// TIA Portal V18 export
FUNCTION "ST10_Output" : Void   // FC1002, LAD
{ S7_Optimized_Access := 'FALSE' }
VERSION : 0.1
// stored: AutoNumber false, IsIECCheckEnabled false, SetENOAutomatically false, UDAEnableTagReadback false
   VAR_TEMP   // added for the SCL form of the ladder/FBD networks
      _w1 : Bool;
      _w2 : Bool;
      _w3 : Bool;
      _w4 : Bool;
      _w5 : Bool;
      _w6 : Bool;
   END_VAR
BEGIN

REGION Network 1 (SCL): 安全门锁定信号映射SafetyDoorCoil
   "oSafetyDoorLocked_1" := "ST10_SysOutput".SafetyDoorCoil[1];
   "oSafetyDoorLocked_2" := "ST10_SysOutput".SafetyDoorCoil[2];
   "oSafetyDoorLocked_3" := "ST10_SysOutput".SafetyDoorCoil[3];
   "oSafetyDoorLocked_4" := "ST10_SysOutput".SafetyDoorCoil[4];
   "oSafetyDoorLocked_5" := "ST10_SysOutput".SafetyDoorCoil[5];
   "oSafetyDoorLocked_6" := "ST10_SysOutput".SafetyDoorCoil[6];
   "oSafetyDoorLocked_7" := "ST10_SysOutput".SafetyDoorCoil[7];
   "oSafetyDoorLocked_8" := "ST10_SysOutput".SafetyDoorCoil[8];
   "oSafetyDoorLocked" := "ST10_SysOutput".SafetyDoorCoil[9];
END_REGION

REGION Network 2 (SCL): 安全门锁定信号映射SafetyDoorCoil
   "oMaterielDoorLocked_H1" := "ST10_SysOutput".MaterialDoorCoil[1];
   "oMaterielDoorLocked_H2" := "ST10_SysOutput".MaterialDoorCoil[2];
   "oMaterielDoorLocked_J1" := "ST10_SysOutput".MaterialDoorCoil[3];
   "oMaterielDoorLocked_J2" := "ST10_SysOutput".MaterialDoorCoil[4];
   "oMaterielDoorLocked_K1" := "ST10_SysOutput".MaterialDoorCoil[5];
   "oMaterielDoorLocked_K2" := "ST10_SysOutput".MaterialDoorCoil[6];
   "oMaterielDoorLocked_L1" := "ST10_SysOutput".MaterialDoorCoil[7];


   "oE-NG-01SafetyGate" := "ST10_SysOutput".MaterialDoorCoil[8];
   "oE-NG-02SafetyGate" := "ST10_SysOutput".MaterialDoorCoil[9];
END_REGION

REGION Network 3: 塔灯
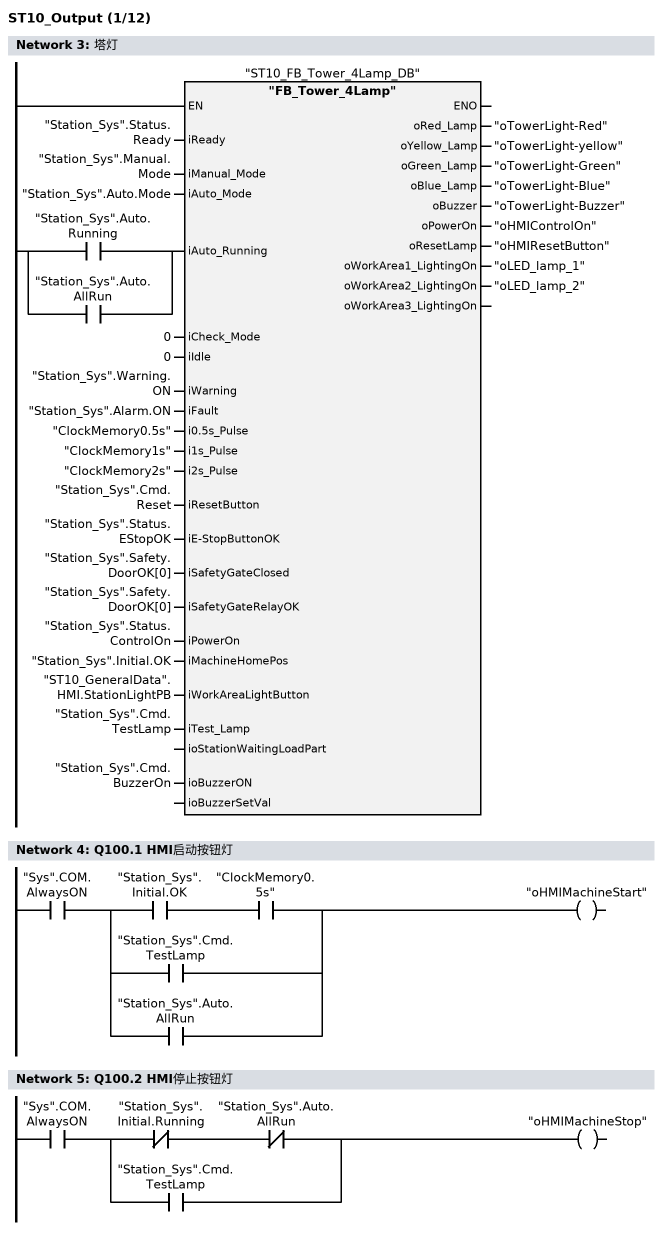
   RUNG wire#powerrail
      "ST10_FB_Tower_4Lamp_DB"(iAuto_Running := wire#w1, iReady := "Station_Sys".Status.Ready, iManual_Mode := "Station_Sys".Manual.Mode, iAuto_Mode := "Station_Sys".Auto.Mode, iCheck_Mode := 0, iIdle := 0, iWarning := "Station_Sys".Warning.ON, iFault := "Station_Sys".Alarm.ON, "i0.5s_Pulse" := "ClockMemory0.5s", i1s_Pulse := "ClockMemory1s", i2s_Pulse := "ClockMemory2s", iResetButton := "Station_Sys".Cmd.Reset, "iE-StopButtonOK" := "Station_Sys".Status.EStopOK, iSafetyGateClosed := "Station_Sys".Safety.DoorOK[0], iSafetyGateRelayOK := "Station_Sys".Safety.DoorOK[0], iPowerOn := "Station_Sys".Status.ControlOn, iMachineHomePos := "Station_Sys".Initial.OK, iWorkAreaLightButton := "ST10_GeneralData".HMI.StationLightPB, iTest_Lamp := "Station_Sys".Cmd.TestLamp, ioStationWaitingLoadPart :=, ioBuzzerON := "Station_Sys".Cmd.BuzzerOn, ioBuzzerSetVal :=, oRed_Lamp => "oTowerLight-Red", oYellow_Lamp => "oTowerLight-yellow", oGreen_Lamp => "oTowerLight-Green", oBlue_Lamp => "oTowerLight-Blue", oBuzzer => "oTowerLight-Buzzer", oPowerOn => "oHMIControlOn", oResetLamp => "oHMIResetButton", oWorkArea1_LightingOn => "oLED_lamp_1", oWorkArea2_LightingOn => "oLED_lamp_2", oWorkArea3_LightingOn =>)
   END_RUNG
   RUNG wire#powerrail
      Contact( "Station_Sys".Auto.Running )
   END_RUNG wire#w1
   RUNG wire#powerrail
      Contact( "Station_Sys".Auto.AllRun )
   END_RUNG wire#w1
   // the same network as SCL:
   "ST10_FB_Tower_4Lamp_DB"(iReady := "Station_Sys".Status.Ready,   // "FB_Tower_4Lamp"
                           iManual_Mode := "Station_Sys".Manual.Mode,
                           iAuto_Mode := "Station_Sys".Auto.Mode,
                           iAuto_Running := "Station_Sys".Auto.Running OR "Station_Sys".Auto.AllRun,
                           iCheck_Mode := 0,
                           iIdle := 0,
                           iWarning := "Station_Sys".Warning.ON,
                           iFault := "Station_Sys".Alarm.ON,
                           "i0.5s_Pulse" := "ClockMemory0.5s",
                           i1s_Pulse := "ClockMemory1s",
                           i2s_Pulse := "ClockMemory2s",
                           iResetButton := "Station_Sys".Cmd.Reset,
                           "iE-StopButtonOK" := "Station_Sys".Status.EStopOK,
                           iSafetyGateClosed := "Station_Sys".Safety.DoorOK[0],
                           iSafetyGateRelayOK := "Station_Sys".Safety.DoorOK[0],
                           iPowerOn := "Station_Sys".Status.ControlOn,
                           iMachineHomePos := "Station_Sys".Initial.OK,
                           iWorkAreaLightButton := "ST10_GeneralData".HMI.StationLightPB,
                           iTest_Lamp := "Station_Sys".Cmd.TestLamp,
                           ioBuzzerON := "Station_Sys".Cmd.BuzzerOn,
                           oRed_Lamp => "oTowerLight-Red",
                           oYellow_Lamp => "oTowerLight-yellow",
                           oGreen_Lamp => "oTowerLight-Green",
                           oBlue_Lamp => "oTowerLight-Blue",
                           oBuzzer => "oTowerLight-Buzzer",
                           oPowerOn => "oHMIControlOn",
                           oResetLamp => "oHMIResetButton",
                           oWorkArea1_LightingOn => "oLED_lamp_1",
                           oWorkArea2_LightingOn => "oLED_lamp_2");
END_REGION

REGION Network 4: Q100.1 HMI启动按钮灯
   RUNG wire#powerrail
      Contact( "Sys".COM.AlwaysON )
      wire#w1
      Contact( "Station_Sys".Initial.OK )
      Contact( "ClockMemory0.5s" )
      wire#w2
      Coil( "oHMIMachineStart" )
   END_RUNG
   RUNG wire#w1
      Contact( "Station_Sys".Cmd.TestLamp )
   END_RUNG wire#w2
   RUNG wire#w1
      Contact( "Station_Sys".Auto.AllRun )
   END_RUNG wire#w2
   // the same network as SCL:
   "oHMIMachineStart" := "Sys".COM.AlwaysON AND (("Station_Sys".Initial.OK AND "ClockMemory0.5s") OR "Station_Sys".Cmd.TestLamp OR "Station_Sys".Auto.AllRun);
END_REGION

REGION Network 5: Q100.2 HMI停止按钮灯
   RUNG wire#powerrail
      Contact( "Sys".COM.AlwaysON )
      wire#w1
      I_Contact( "Station_Sys".Initial.Running )
      I_Contact( "Station_Sys".Auto.AllRun )
      wire#w2
      Coil( "oHMIMachineStop" )
   END_RUNG
   RUNG wire#w1
      Contact( "Station_Sys".Cmd.TestLamp )
   END_RUNG wire#w2
   // the same network as SCL:
   "oHMIMachineStop" := "Sys".COM.AlwaysON AND ((NOT "Station_Sys".Initial.Running AND NOT "Station_Sys".Auto.AllRun) OR "Station_Sys".Cmd.TestLamp);
END_REGION

REGION Network 6: Q100.4 HMI开门按钮灯
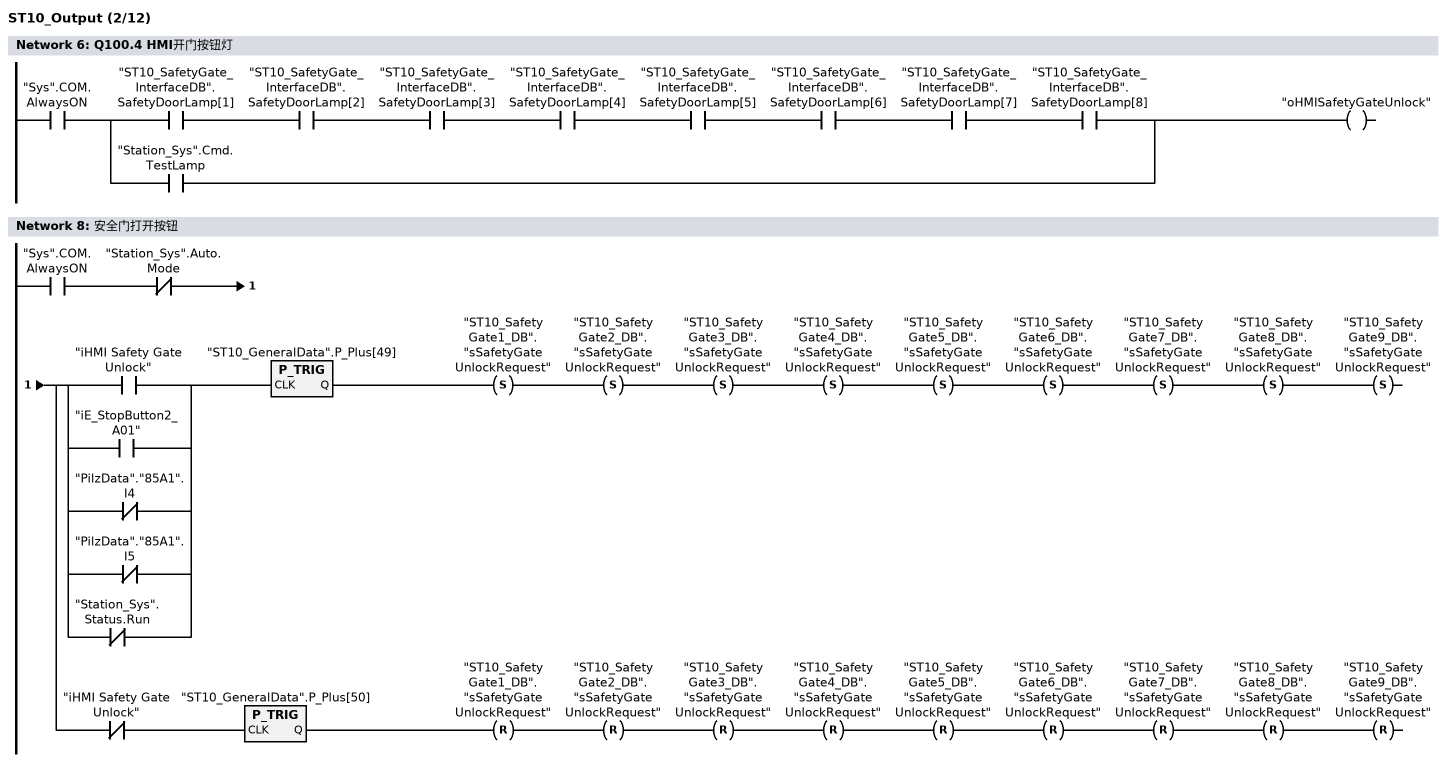
   RUNG wire#powerrail
      Contact( "Sys".COM.AlwaysON )
      wire#w1
      Contact( "ST10_SafetyGate_InterfaceDB".SafetyDoorLamp[1] )
      Contact( "ST10_SafetyGate_InterfaceDB".SafetyDoorLamp[2] )
      Contact( "ST10_SafetyGate_InterfaceDB".SafetyDoorLamp[3] )
      Contact( "ST10_SafetyGate_InterfaceDB".SafetyDoorLamp[4] )
      Contact( "ST10_SafetyGate_InterfaceDB".SafetyDoorLamp[5] )
      Contact( "ST10_SafetyGate_InterfaceDB".SafetyDoorLamp[6] )
      Contact( "ST10_SafetyGate_InterfaceDB".SafetyDoorLamp[7] )
      Contact( "ST10_SafetyGate_InterfaceDB".SafetyDoorLamp[8] )
      wire#w2
      Coil( "oHMISafetyGateUnlock" )
   END_RUNG
   RUNG wire#w1
      Contact( "Station_Sys".Cmd.TestLamp )
   END_RUNG wire#w2
   // the same network as SCL:
   "oHMISafetyGateUnlock" := "Sys".COM.AlwaysON AND (("ST10_SafetyGate_InterfaceDB".SafetyDoorLamp[1] AND "ST10_SafetyGate_InterfaceDB".SafetyDoorLamp[2] AND "ST10_SafetyGate_InterfaceDB".SafetyDoorLamp[3] AND "ST10_SafetyGate_InterfaceDB".SafetyDoorLamp[4] AND "ST10_SafetyGate_InterfaceDB".SafetyDoorLamp[5] AND "ST10_SafetyGate_InterfaceDB".SafetyDoorLamp[6] AND "ST10_SafetyGate_InterfaceDB".SafetyDoorLamp[7] AND "ST10_SafetyGate_InterfaceDB".SafetyDoorLamp[8]) OR "Station_Sys".Cmd.TestLamp);
END_REGION

REGION Network 8: 安全门打开按钮
   RUNG wire#powerrail
      Contact( "Sys".COM.AlwaysON )
      I_Contact( "Station_Sys".Auto.Mode )
      wire#w1
      Contact( "iHMI Safety Gate Unlock" )
      wire#w2
      P_Trig( "ST10_GeneralData".P_Plus[49] )
      S_Coil( "ST10_SafetyGate1_DB"."sSafetyGate UnlockRequest" )
      S_Coil( "ST10_SafetyGate2_DB"."sSafetyGate UnlockRequest" )
      S_Coil( "ST10_SafetyGate3_DB"."sSafetyGate UnlockRequest" )
      S_Coil( "ST10_SafetyGate4_DB"."sSafetyGate UnlockRequest" )
      S_Coil( "ST10_SafetyGate5_DB"."sSafetyGate UnlockRequest" )
      S_Coil( "ST10_SafetyGate6_DB"."sSafetyGate UnlockRequest" )
      S_Coil( "ST10_SafetyGate7_DB"."sSafetyGate UnlockRequest" )
      S_Coil( "ST10_SafetyGate8_DB"."sSafetyGate UnlockRequest" )
      S_Coil( "ST10_SafetyGate9_DB"."sSafetyGate UnlockRequest" )
   END_RUNG
   RUNG wire#w1
      Contact( "iE_StopButton2_A01" )
   END_RUNG wire#w2
   RUNG wire#w1
      I_Contact( "PilzData"."85A1".I4 )
   END_RUNG wire#w2
   RUNG wire#w1
      I_Contact( "PilzData"."85A1".I5 )
   END_RUNG wire#w2
   RUNG wire#w1
      I_Contact( "Station_Sys".Status.Run )
   END_RUNG wire#w2
   RUNG wire#w1
      I_Contact( "iHMI Safety Gate Unlock" )
      P_Trig( "ST10_GeneralData".P_Plus[50] )
      R_Coil( "ST10_SafetyGate1_DB"."sSafetyGate UnlockRequest" )
      R_Coil( "ST10_SafetyGate2_DB"."sSafetyGate UnlockRequest" )
      R_Coil( "ST10_SafetyGate3_DB"."sSafetyGate UnlockRequest" )
      R_Coil( "ST10_SafetyGate4_DB"."sSafetyGate UnlockRequest" )
      R_Coil( "ST10_SafetyGate5_DB"."sSafetyGate UnlockRequest" )
      R_Coil( "ST10_SafetyGate6_DB"."sSafetyGate UnlockRequest" )
      R_Coil( "ST10_SafetyGate7_DB"."sSafetyGate UnlockRequest" )
      R_Coil( "ST10_SafetyGate8_DB"."sSafetyGate UnlockRequest" )
      R_Coil( "ST10_SafetyGate9_DB"."sSafetyGate UnlockRequest" )
   END_RUNG
   // the same network as SCL:
   #_w1 := "Sys".COM.AlwaysON AND NOT "Station_Sys".Auto.Mode;
   #_w2 := #_w1 AND ("iHMI Safety Gate Unlock" OR "iE_StopButton2_A01" OR NOT "PilzData"."85A1".I4 OR NOT "PilzData"."85A1".I5 OR NOT "Station_Sys".Status.Run);
   #_w3 := #_w2 AND NOT "ST10_GeneralData".P_Plus[49];   // rising edge
   "ST10_GeneralData".P_Plus[49] := #_w2;
   IF #_w3 THEN
       "ST10_SafetyGate1_DB"."sSafetyGate UnlockRequest" := TRUE;
       "ST10_SafetyGate2_DB"."sSafetyGate UnlockRequest" := TRUE;
       "ST10_SafetyGate3_DB"."sSafetyGate UnlockRequest" := TRUE;
       "ST10_SafetyGate4_DB"."sSafetyGate UnlockRequest" := TRUE;
       "ST10_SafetyGate5_DB"."sSafetyGate UnlockRequest" := TRUE;
       "ST10_SafetyGate6_DB"."sSafetyGate UnlockRequest" := TRUE;
       "ST10_SafetyGate7_DB"."sSafetyGate UnlockRequest" := TRUE;
       "ST10_SafetyGate8_DB"."sSafetyGate UnlockRequest" := TRUE;
       "ST10_SafetyGate9_DB"."sSafetyGate UnlockRequest" := TRUE;
   END_IF;
   #_w4 := #_w1 AND NOT "iHMI Safety Gate Unlock";
   #_w5 := #_w4 AND NOT "ST10_GeneralData".P_Plus[50];   // rising edge
   "ST10_GeneralData".P_Plus[50] := #_w4;
   IF #_w5 THEN
       "ST10_SafetyGate1_DB"."sSafetyGate UnlockRequest" := FALSE;
       "ST10_SafetyGate2_DB"."sSafetyGate UnlockRequest" := FALSE;
       "ST10_SafetyGate3_DB"."sSafetyGate UnlockRequest" := FALSE;
       "ST10_SafetyGate4_DB"."sSafetyGate UnlockRequest" := FALSE;
       "ST10_SafetyGate5_DB"."sSafetyGate UnlockRequest" := FALSE;
       "ST10_SafetyGate6_DB"."sSafetyGate UnlockRequest" := FALSE;
       "ST10_SafetyGate7_DB"."sSafetyGate UnlockRequest" := FALSE;
       "ST10_SafetyGate8_DB"."sSafetyGate UnlockRequest" := FALSE;
       "ST10_SafetyGate9_DB"."sSafetyGate UnlockRequest" := FALSE;
   END_IF;
END_REGION

REGION Network 9: 安全门关闭
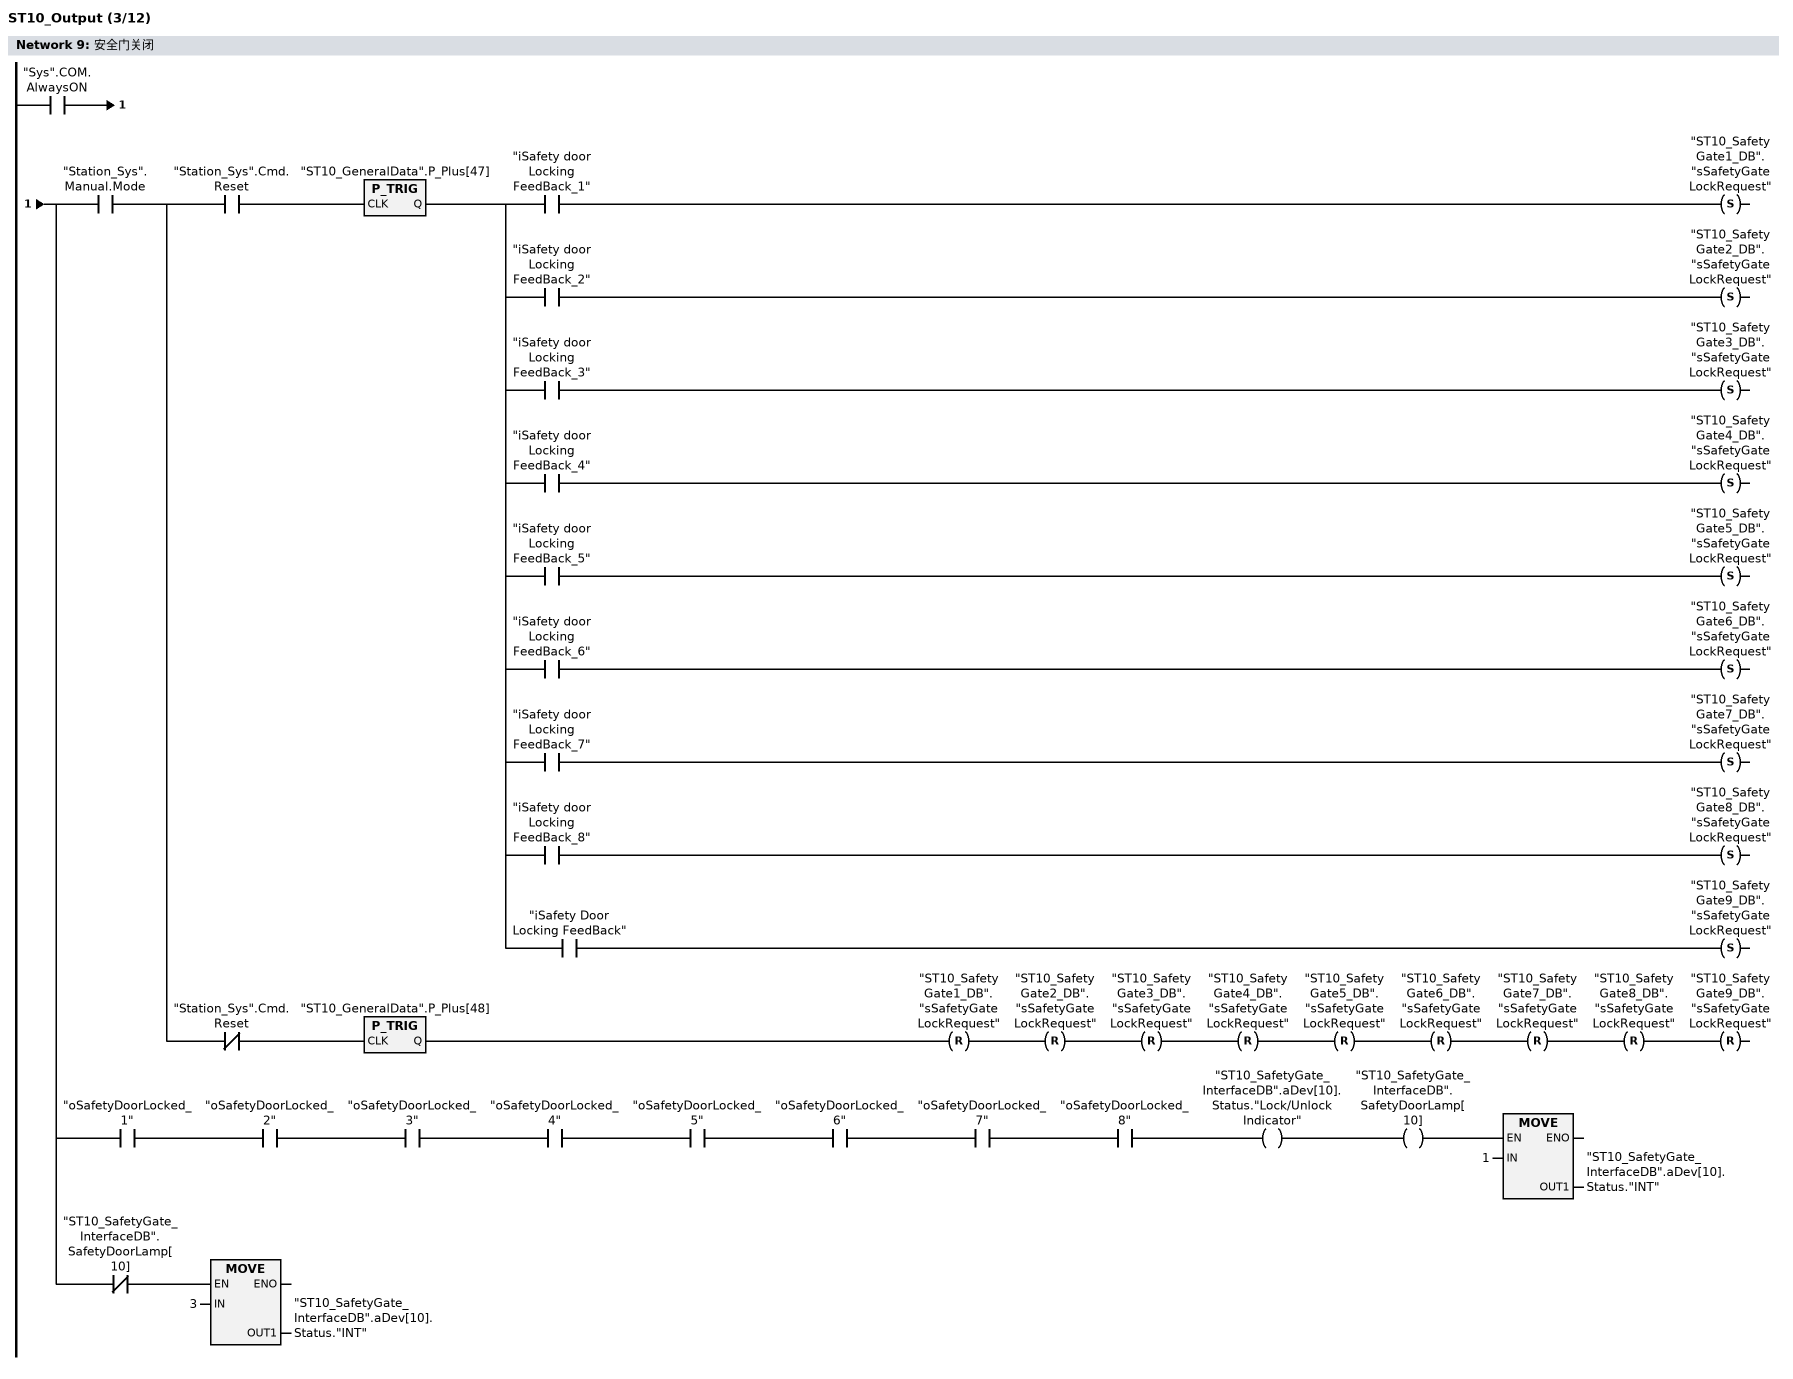
   RUNG wire#powerrail
      Contact( "Sys".COM.AlwaysON )
      wire#w1
      Contact( "Station_Sys".Manual.Mode )
      wire#w2
      Contact( "Station_Sys".Cmd.Reset )
      P_Trig( "ST10_GeneralData".P_Plus[47] )
      wire#w3
      Contact( "iSafety door Locking FeedBack_1" )
      S_Coil( "ST10_SafetyGate1_DB"."sSafetyGate LockRequest" )
   END_RUNG
   RUNG wire#w3
      Contact( "iSafety door Locking FeedBack_2" )
      S_Coil( "ST10_SafetyGate2_DB"."sSafetyGate LockRequest" )
   END_RUNG
   RUNG wire#w3
      Contact( "iSafety door Locking FeedBack_3" )
      S_Coil( "ST10_SafetyGate3_DB"."sSafetyGate LockRequest" )
   END_RUNG
   RUNG wire#w3
      Contact( "iSafety door Locking FeedBack_4" )
      S_Coil( "ST10_SafetyGate4_DB"."sSafetyGate LockRequest" )
   END_RUNG
   RUNG wire#w3
      Contact( "iSafety door Locking FeedBack_5" )
      S_Coil( "ST10_SafetyGate5_DB"."sSafetyGate LockRequest" )
   END_RUNG
   RUNG wire#w3
      Contact( "iSafety door Locking FeedBack_6" )
      S_Coil( "ST10_SafetyGate6_DB"."sSafetyGate LockRequest" )
   END_RUNG
   RUNG wire#w3
      Contact( "iSafety door Locking FeedBack_7" )
      S_Coil( "ST10_SafetyGate7_DB"."sSafetyGate LockRequest" )
   END_RUNG
   RUNG wire#w3
      Contact( "iSafety door Locking FeedBack_8" )
      S_Coil( "ST10_SafetyGate8_DB"."sSafetyGate LockRequest" )
   END_RUNG
   RUNG wire#w3
      Contact( "iSafety Door Locking FeedBack" )
      S_Coil( "ST10_SafetyGate9_DB"."sSafetyGate LockRequest" )
   END_RUNG
   RUNG wire#w2
      I_Contact( "Station_Sys".Cmd.Reset )
      P_Trig( "ST10_GeneralData".P_Plus[48] )
      R_Coil( "ST10_SafetyGate1_DB"."sSafetyGate LockRequest" )
      R_Coil( "ST10_SafetyGate2_DB"."sSafetyGate LockRequest" )
      R_Coil( "ST10_SafetyGate3_DB"."sSafetyGate LockRequest" )
      R_Coil( "ST10_SafetyGate4_DB"."sSafetyGate LockRequest" )
      R_Coil( "ST10_SafetyGate5_DB"."sSafetyGate LockRequest" )
      R_Coil( "ST10_SafetyGate6_DB"."sSafetyGate LockRequest" )
      R_Coil( "ST10_SafetyGate7_DB"."sSafetyGate LockRequest" )
      R_Coil( "ST10_SafetyGate8_DB"."sSafetyGate LockRequest" )
      R_Coil( "ST10_SafetyGate9_DB"."sSafetyGate LockRequest" )
   END_RUNG
   RUNG wire#w1
      Contact( "oSafetyDoorLocked_1" )
      Contact( "oSafetyDoorLocked_2" )
      Contact( "oSafetyDoorLocked_3" )
      Contact( "oSafetyDoorLocked_4" )
      Contact( "oSafetyDoorLocked_5" )
      Contact( "oSafetyDoorLocked_6" )
      Contact( "oSafetyDoorLocked_7" )
      Contact( "oSafetyDoorLocked_8" )
      Coil( "ST10_SafetyGate_InterfaceDB".aDev[10].Status."Lock/Unlock Indicator" )
      Coil( "ST10_SafetyGate_InterfaceDB".SafetyDoorLamp[10] )
      Move(in := 1, out1 => "ST10_SafetyGate_InterfaceDB".aDev[10].Status."INT")
   END_RUNG
   RUNG wire#w1
      I_Contact( "ST10_SafetyGate_InterfaceDB".SafetyDoorLamp[10] )
      Move(in := 3, out1 => "ST10_SafetyGate_InterfaceDB".aDev[10].Status."INT")
   END_RUNG
   // the same network as SCL:
   #_w1 := "Sys".COM.AlwaysON AND "Station_Sys".Manual.Mode;
   #_w2 := #_w1 AND "Station_Sys".Cmd.Reset;
   #_w3 := #_w2 AND NOT "ST10_GeneralData".P_Plus[47];   // rising edge
   "ST10_GeneralData".P_Plus[47] := #_w2;
   IF #_w3 AND "iSafety door Locking FeedBack_1" THEN
       "ST10_SafetyGate1_DB"."sSafetyGate LockRequest" := TRUE;
   END_IF;
   IF #_w3 AND "iSafety door Locking FeedBack_2" THEN
       "ST10_SafetyGate2_DB"."sSafetyGate LockRequest" := TRUE;
   END_IF;
   IF #_w3 AND "iSafety door Locking FeedBack_3" THEN
       "ST10_SafetyGate3_DB"."sSafetyGate LockRequest" := TRUE;
   END_IF;
   IF #_w3 AND "iSafety door Locking FeedBack_4" THEN
       "ST10_SafetyGate4_DB"."sSafetyGate LockRequest" := TRUE;
   END_IF;
   IF #_w3 AND "iSafety door Locking FeedBack_5" THEN
       "ST10_SafetyGate5_DB"."sSafetyGate LockRequest" := TRUE;
   END_IF;
   IF #_w3 AND "iSafety door Locking FeedBack_6" THEN
       "ST10_SafetyGate6_DB"."sSafetyGate LockRequest" := TRUE;
   END_IF;
   IF #_w3 AND "iSafety door Locking FeedBack_7" THEN
       "ST10_SafetyGate7_DB"."sSafetyGate LockRequest" := TRUE;
   END_IF;
   IF #_w3 AND "iSafety door Locking FeedBack_8" THEN
       "ST10_SafetyGate8_DB"."sSafetyGate LockRequest" := TRUE;
   END_IF;
   IF #_w3 AND "iSafety Door Locking FeedBack" THEN
       "ST10_SafetyGate9_DB"."sSafetyGate LockRequest" := TRUE;
   END_IF;
   #_w4 := #_w1 AND NOT "Station_Sys".Cmd.Reset;
   #_w5 := #_w4 AND NOT "ST10_GeneralData".P_Plus[48];   // rising edge
   "ST10_GeneralData".P_Plus[48] := #_w4;
   IF #_w5 THEN
       "ST10_SafetyGate1_DB"."sSafetyGate LockRequest" := FALSE;
       "ST10_SafetyGate2_DB"."sSafetyGate LockRequest" := FALSE;
       "ST10_SafetyGate3_DB"."sSafetyGate LockRequest" := FALSE;
       "ST10_SafetyGate4_DB"."sSafetyGate LockRequest" := FALSE;
       "ST10_SafetyGate5_DB"."sSafetyGate LockRequest" := FALSE;
       "ST10_SafetyGate6_DB"."sSafetyGate LockRequest" := FALSE;
       "ST10_SafetyGate7_DB"."sSafetyGate LockRequest" := FALSE;
       "ST10_SafetyGate8_DB"."sSafetyGate LockRequest" := FALSE;
       "ST10_SafetyGate9_DB"."sSafetyGate LockRequest" := FALSE;
   END_IF;
   "ST10_SafetyGate_InterfaceDB".aDev[10].Status."Lock/Unlock Indicator" := "Sys".COM.AlwaysON AND "oSafetyDoorLocked_1" AND "oSafetyDoorLocked_2" AND "oSafetyDoorLocked_3" AND "oSafetyDoorLocked_4" AND "oSafetyDoorLocked_5" AND "oSafetyDoorLocked_6" AND "oSafetyDoorLocked_7" AND "oSafetyDoorLocked_8";
   "ST10_SafetyGate_InterfaceDB".SafetyDoorLamp[10] := "Sys".COM.AlwaysON AND "oSafetyDoorLocked_1" AND "oSafetyDoorLocked_2" AND "oSafetyDoorLocked_3" AND "oSafetyDoorLocked_4" AND "oSafetyDoorLocked_5" AND "oSafetyDoorLocked_6" AND "oSafetyDoorLocked_7" AND "oSafetyDoorLocked_8";
   IF "Sys".COM.AlwaysON AND "oSafetyDoorLocked_1" AND "oSafetyDoorLocked_2" AND "oSafetyDoorLocked_3" AND "oSafetyDoorLocked_4" AND "oSafetyDoorLocked_5" AND "oSafetyDoorLocked_6" AND "oSafetyDoorLocked_7" AND "oSafetyDoorLocked_8" THEN
       "ST10_SafetyGate_InterfaceDB".aDev[10].Status."INT" := 1;
   END_IF;
   IF "Sys".COM.AlwaysON AND NOT "ST10_SafetyGate_InterfaceDB".SafetyDoorLamp[10] THEN
       "ST10_SafetyGate_InterfaceDB".aDev[10].Status."INT" := 3;
   END_IF;
END_REGION

REGION Network 11: E-NG料盒-01安全门锁按钮灯
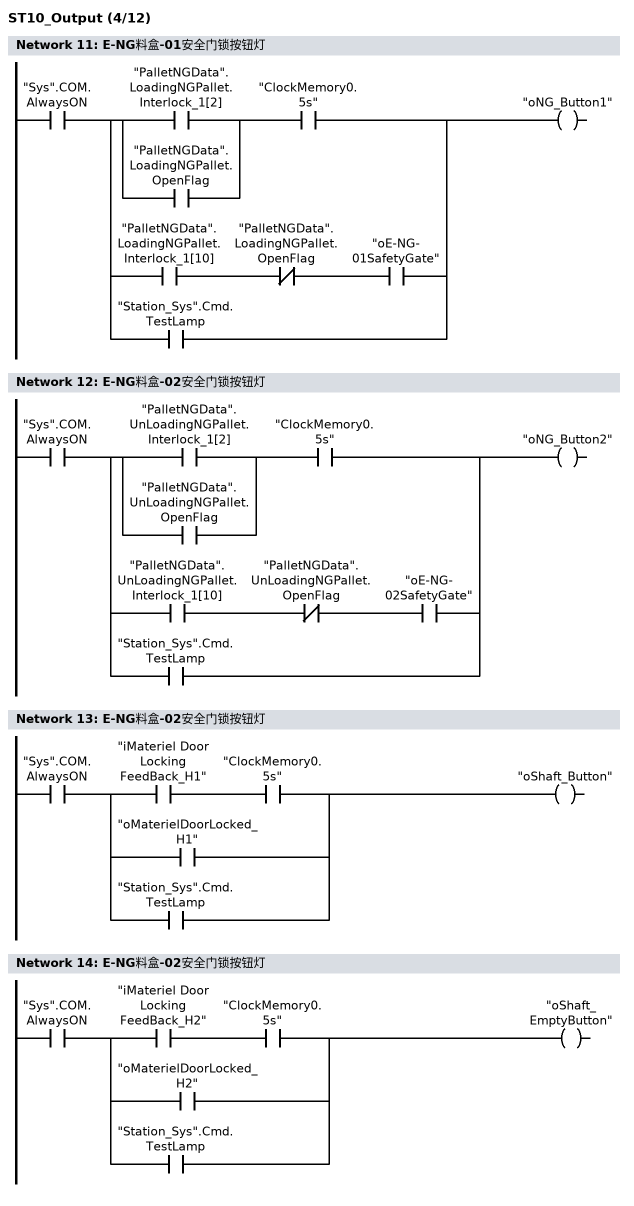
   RUNG wire#powerrail
      Contact( "Sys".COM.AlwaysON )
      wire#w1
      Contact( "PalletNGData".LoadingNGPallet.Interlock_1[2] )
      wire#w2
      Contact( "ClockMemory0.5s" )
      wire#w3
      Coil( "oNG_Button1" )
   END_RUNG
   RUNG wire#w1
      Contact( "PalletNGData".LoadingNGPallet.OpenFlag )
   END_RUNG wire#w2
   RUNG wire#w1
      Contact( "PalletNGData".LoadingNGPallet.Interlock_1[10] )
      I_Contact( "PalletNGData".LoadingNGPallet.OpenFlag )
      Contact( "oE-NG-01SafetyGate" )
   END_RUNG wire#w3
   RUNG wire#w1
      Contact( "Station_Sys".Cmd.TestLamp )
   END_RUNG wire#w3
   // the same network as SCL:
   "oNG_Button1" := "Sys".COM.AlwaysON AND ((("PalletNGData".LoadingNGPallet.Interlock_1[2] OR "PalletNGData".LoadingNGPallet.OpenFlag) AND "ClockMemory0.5s") OR ("PalletNGData".LoadingNGPallet.Interlock_1[10] AND NOT "PalletNGData".LoadingNGPallet.OpenFlag AND "oE-NG-01SafetyGate") OR "Station_Sys".Cmd.TestLamp);
END_REGION

REGION Network 12: E-NG料盒-02安全门锁按钮灯
   RUNG wire#powerrail
      Contact( "Sys".COM.AlwaysON )
      wire#w1
      Contact( "PalletNGData".UnLoadingNGPallet.Interlock_1[2] )
      wire#w2
      Contact( "ClockMemory0.5s" )
      wire#w3
      Coil( "oNG_Button2" )
   END_RUNG
   RUNG wire#w1
      Contact( "PalletNGData".UnLoadingNGPallet.OpenFlag )
   END_RUNG wire#w2
   RUNG wire#w1
      Contact( "PalletNGData".UnLoadingNGPallet.Interlock_1[10] )
      I_Contact( "PalletNGData".UnLoadingNGPallet.OpenFlag )
      Contact( "oE-NG-02SafetyGate" )
   END_RUNG wire#w3
   RUNG wire#w1
      Contact( "Station_Sys".Cmd.TestLamp )
   END_RUNG wire#w3
   // the same network as SCL:
   "oNG_Button2" := "Sys".COM.AlwaysON AND ((("PalletNGData".UnLoadingNGPallet.Interlock_1[2] OR "PalletNGData".UnLoadingNGPallet.OpenFlag) AND "ClockMemory0.5s") OR ("PalletNGData".UnLoadingNGPallet.Interlock_1[10] AND NOT "PalletNGData".UnLoadingNGPallet.OpenFlag AND "oE-NG-02SafetyGate") OR "Station_Sys".Cmd.TestLamp);
END_REGION

REGION Network 13: E-NG料盒-02安全门锁按钮灯
   RUNG wire#powerrail
      Contact( "Sys".COM.AlwaysON )
      wire#w1
      Contact( "iMateriel Door Locking FeedBack_H1" )
      Contact( "ClockMemory0.5s" )
      wire#w2
      Coil( "oShaft_Button" )
   END_RUNG
   RUNG wire#w1
      Contact( "oMaterielDoorLocked_H1" )
   END_RUNG wire#w2
   RUNG wire#w1
      Contact( "Station_Sys".Cmd.TestLamp )
   END_RUNG wire#w2
   // the same network as SCL:
   "oShaft_Button" := "Sys".COM.AlwaysON AND (("iMateriel Door Locking FeedBack_H1" AND "ClockMemory0.5s") OR "oMaterielDoorLocked_H1" OR "Station_Sys".Cmd.TestLamp);
END_REGION

REGION Network 14: E-NG料盒-02安全门锁按钮灯
   RUNG wire#powerrail
      Contact( "Sys".COM.AlwaysON )
      wire#w1
      Contact( "iMateriel Door Locking FeedBack_H2" )
      Contact( "ClockMemory0.5s" )
      wire#w2
      Coil( "oShaft_EmptyButton" )
   END_RUNG
   RUNG wire#w1
      Contact( "oMaterielDoorLocked_H2" )
   END_RUNG wire#w2
   RUNG wire#w1
      Contact( "Station_Sys".Cmd.TestLamp )
   END_RUNG wire#w2
   // the same network as SCL:
   "oShaft_EmptyButton" := "Sys".COM.AlwaysON AND (("iMateriel Door Locking FeedBack_H2" AND "ClockMemory0.5s") OR "oMaterielDoorLocked_H2" OR "Station_Sys".Cmd.TestLamp);
END_REGION

REGION Network 15: E-NG料盒-02安全门锁按钮灯
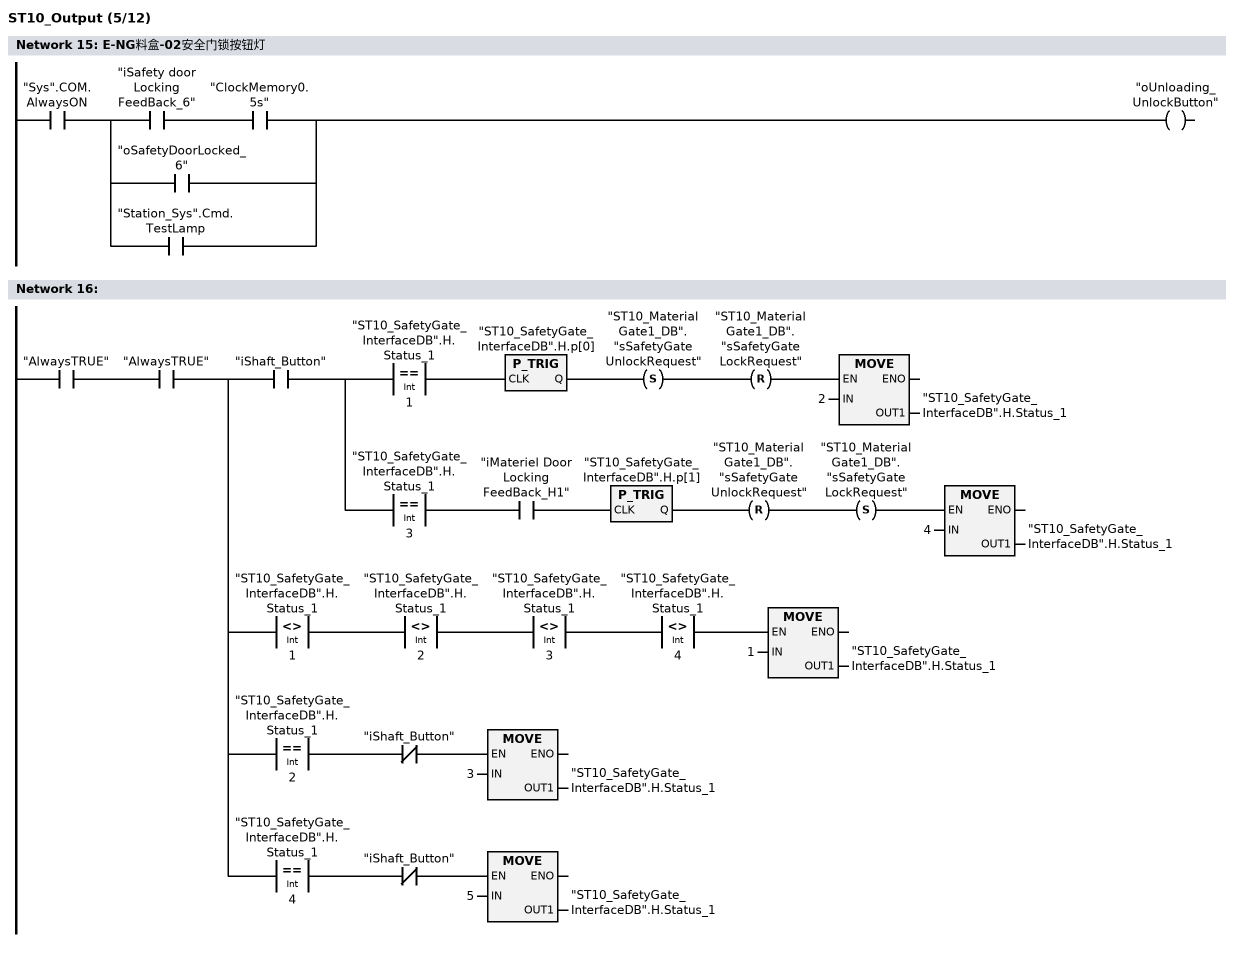
   RUNG wire#powerrail
      Contact( "Sys".COM.AlwaysON )
      wire#w1
      Contact( "iSafety door Locking FeedBack_6" )
      Contact( "ClockMemory0.5s" )
      wire#w2
      Coil( "oUnloading_UnlockButton" )
   END_RUNG
   RUNG wire#w1
      Contact( "oSafetyDoorLocked_6" )
   END_RUNG wire#w2
   RUNG wire#w1
      Contact( "Station_Sys".Cmd.TestLamp )
   END_RUNG wire#w2
   // the same network as SCL:
   "oUnloading_UnlockButton" := "Sys".COM.AlwaysON AND (("iSafety door Locking FeedBack_6" AND "ClockMemory0.5s") OR "oSafetyDoorLocked_6" OR "Station_Sys".Cmd.TestLamp);
END_REGION

REGION Network 16
   RUNG wire#powerrail
      Contact( "AlwaysTRUE" )
      Contact( "AlwaysTRUE" )
      wire#w1
      Contact( "iShaft_Button" )
      wire#w2
      { S7_Templates := "SrcType := Int" } EQ_Contact(in1 := "ST10_SafetyGate_InterfaceDB".H.Status_1, in2 := 1)
      P_Trig( "ST10_SafetyGate_InterfaceDB".H.p[0] )
      S_Coil( "ST10_MaterialGate1_DB"."sSafetyGate UnlockRequest" )
      R_Coil( "ST10_MaterialGate1_DB"."sSafetyGate LockRequest" )
      Move(in := 2, out1 => "ST10_SafetyGate_InterfaceDB".H.Status_1)
   END_RUNG
   RUNG wire#w2
      { S7_Templates := "SrcType := Int" } EQ_Contact(in1 := "ST10_SafetyGate_InterfaceDB".H.Status_1, in2 := 3)
      Contact( "iMateriel Door Locking FeedBack_H1" )
      P_Trig( "ST10_SafetyGate_InterfaceDB".H.p[1] )
      R_Coil( "ST10_MaterialGate1_DB"."sSafetyGate UnlockRequest" )
      S_Coil( "ST10_MaterialGate1_DB"."sSafetyGate LockRequest" )
      Move(in := 4, out1 => "ST10_SafetyGate_InterfaceDB".H.Status_1)
   END_RUNG
   RUNG wire#w1
      { S7_Templates := "SrcType := Int" } NE_Contact(in1 := "ST10_SafetyGate_InterfaceDB".H.Status_1, in2 := 1)
      { S7_Templates := "SrcType := Int" } NE_Contact(in1 := "ST10_SafetyGate_InterfaceDB".H.Status_1, in2 := 2)
      { S7_Templates := "SrcType := Int" } NE_Contact(in1 := "ST10_SafetyGate_InterfaceDB".H.Status_1, in2 := 3)
      { S7_Templates := "SrcType := Int" } NE_Contact(in1 := "ST10_SafetyGate_InterfaceDB".H.Status_1, in2 := 4)
      Move(in := 1, out1 => "ST10_SafetyGate_InterfaceDB".H.Status_1)
   END_RUNG
   RUNG wire#w1
      { S7_Templates := "SrcType := Int" } EQ_Contact(in1 := "ST10_SafetyGate_InterfaceDB".H.Status_1, in2 := 2)
      I_Contact( "iShaft_Button" )
      Move(in := 3, out1 => "ST10_SafetyGate_InterfaceDB".H.Status_1)
   END_RUNG
   RUNG wire#w1
      { S7_Templates := "SrcType := Int" } EQ_Contact(in1 := "ST10_SafetyGate_InterfaceDB".H.Status_1, in2 := 4)
      I_Contact( "iShaft_Button" )
      Move(in := 5, out1 => "ST10_SafetyGate_InterfaceDB".H.Status_1)
   END_RUNG
   // the same network as SCL:
   #_w1 := "AlwaysTRUE" AND "AlwaysTRUE";
   #_w2 := #_w1 AND "iShaft_Button";
   #_w3 := #_w2 AND ("ST10_SafetyGate_InterfaceDB".H.Status_1 = 1);
   #_w4 := #_w3 AND NOT "ST10_SafetyGate_InterfaceDB".H.p[0];   // rising edge
   "ST10_SafetyGate_InterfaceDB".H.p[0] := #_w3;
   IF #_w4 THEN
       "ST10_MaterialGate1_DB"."sSafetyGate UnlockRequest" := TRUE;
       "ST10_MaterialGate1_DB"."sSafetyGate LockRequest" := FALSE;
       "ST10_SafetyGate_InterfaceDB".H.Status_1 := 2;
   END_IF;
   #_w5 := #_w2 AND ("ST10_SafetyGate_InterfaceDB".H.Status_1 = 3) AND "iMateriel Door Locking FeedBack_H1";
   #_w6 := #_w5 AND NOT "ST10_SafetyGate_InterfaceDB".H.p[1];   // rising edge
   "ST10_SafetyGate_InterfaceDB".H.p[1] := #_w5;
   IF #_w6 THEN
       "ST10_MaterialGate1_DB"."sSafetyGate UnlockRequest" := FALSE;
       "ST10_MaterialGate1_DB"."sSafetyGate LockRequest" := TRUE;
       "ST10_SafetyGate_InterfaceDB".H.Status_1 := 4;
   END_IF;
   IF #_w1 AND ("ST10_SafetyGate_InterfaceDB".H.Status_1 <> 1) AND ("ST10_SafetyGate_InterfaceDB".H.Status_1 <> 2) AND ("ST10_SafetyGate_InterfaceDB".H.Status_1 <> 3) AND ("ST10_SafetyGate_InterfaceDB".H.Status_1 <> 4) THEN
       "ST10_SafetyGate_InterfaceDB".H.Status_1 := 1;
   END_IF;
   IF #_w1 AND ("ST10_SafetyGate_InterfaceDB".H.Status_1 = 2) AND NOT "iShaft_Button" THEN
       "ST10_SafetyGate_InterfaceDB".H.Status_1 := 3;
   END_IF;
   IF #_w1 AND ("ST10_SafetyGate_InterfaceDB".H.Status_1 = 4) AND NOT "iShaft_Button" THEN
       "ST10_SafetyGate_InterfaceDB".H.Status_1 := 5;
   END_IF;
END_REGION

REGION Network 17
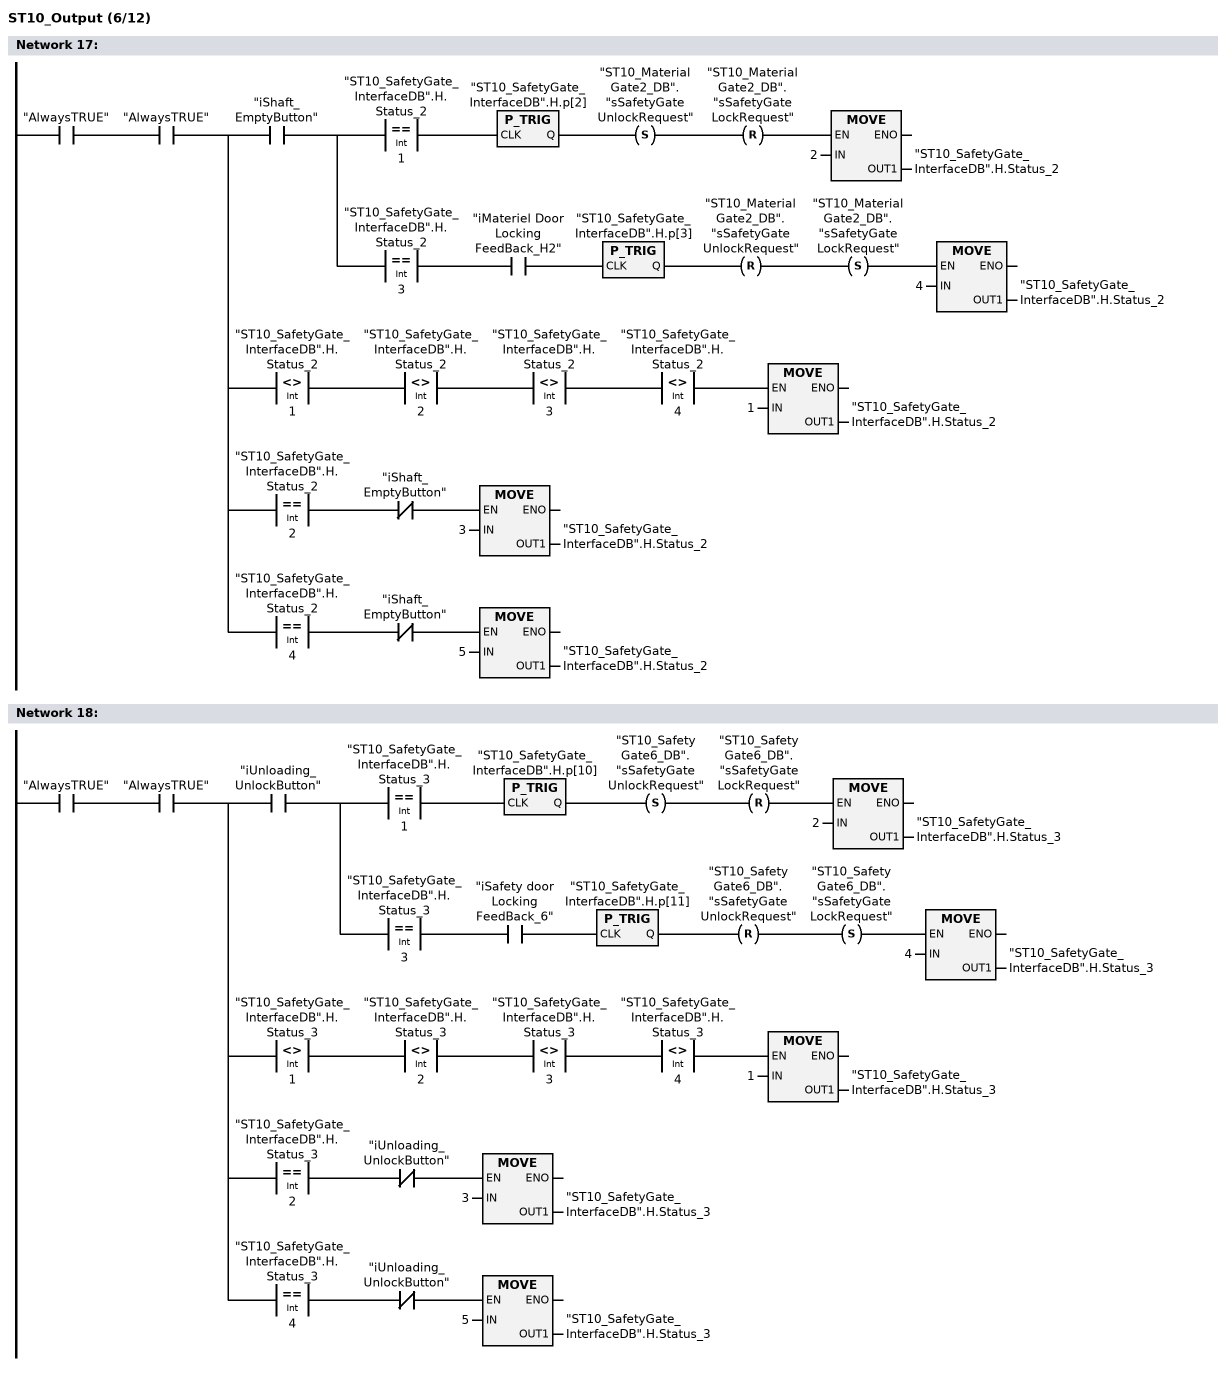
   RUNG wire#powerrail
      Contact( "AlwaysTRUE" )
      Contact( "AlwaysTRUE" )
      wire#w1
      Contact( "iShaft_EmptyButton" )
      wire#w2
      { S7_Templates := "SrcType := Int" } EQ_Contact(in1 := "ST10_SafetyGate_InterfaceDB".H.Status_2, in2 := 1)
      P_Trig( "ST10_SafetyGate_InterfaceDB".H.p[2] )
      S_Coil( "ST10_MaterialGate2_DB"."sSafetyGate UnlockRequest" )
      R_Coil( "ST10_MaterialGate2_DB"."sSafetyGate LockRequest" )
      Move(in := 2, out1 => "ST10_SafetyGate_InterfaceDB".H.Status_2)
   END_RUNG
   RUNG wire#w2
      { S7_Templates := "SrcType := Int" } EQ_Contact(in1 := "ST10_SafetyGate_InterfaceDB".H.Status_2, in2 := 3)
      Contact( "iMateriel Door Locking FeedBack_H2" )
      P_Trig( "ST10_SafetyGate_InterfaceDB".H.p[3] )
      R_Coil( "ST10_MaterialGate2_DB"."sSafetyGate UnlockRequest" )
      S_Coil( "ST10_MaterialGate2_DB"."sSafetyGate LockRequest" )
      Move(in := 4, out1 => "ST10_SafetyGate_InterfaceDB".H.Status_2)
   END_RUNG
   RUNG wire#w1
      { S7_Templates := "SrcType := Int" } NE_Contact(in1 := "ST10_SafetyGate_InterfaceDB".H.Status_2, in2 := 1)
      { S7_Templates := "SrcType := Int" } NE_Contact(in1 := "ST10_SafetyGate_InterfaceDB".H.Status_2, in2 := 2)
      { S7_Templates := "SrcType := Int" } NE_Contact(in1 := "ST10_SafetyGate_InterfaceDB".H.Status_2, in2 := 3)
      { S7_Templates := "SrcType := Int" } NE_Contact(in1 := "ST10_SafetyGate_InterfaceDB".H.Status_2, in2 := 4)
      Move(in := 1, out1 => "ST10_SafetyGate_InterfaceDB".H.Status_2)
   END_RUNG
   RUNG wire#w1
      { S7_Templates := "SrcType := Int" } EQ_Contact(in1 := "ST10_SafetyGate_InterfaceDB".H.Status_2, in2 := 2)
      I_Contact( "iShaft_EmptyButton" )
      Move(in := 3, out1 => "ST10_SafetyGate_InterfaceDB".H.Status_2)
   END_RUNG
   RUNG wire#w1
      { S7_Templates := "SrcType := Int" } EQ_Contact(in1 := "ST10_SafetyGate_InterfaceDB".H.Status_2, in2 := 4)
      I_Contact( "iShaft_EmptyButton" )
      Move(in := 5, out1 => "ST10_SafetyGate_InterfaceDB".H.Status_2)
   END_RUNG
   // the same network as SCL:
   #_w1 := "AlwaysTRUE" AND "AlwaysTRUE";
   #_w2 := #_w1 AND "iShaft_EmptyButton";
   #_w3 := #_w2 AND ("ST10_SafetyGate_InterfaceDB".H.Status_2 = 1);
   #_w4 := #_w3 AND NOT "ST10_SafetyGate_InterfaceDB".H.p[2];   // rising edge
   "ST10_SafetyGate_InterfaceDB".H.p[2] := #_w3;
   IF #_w4 THEN
       "ST10_MaterialGate2_DB"."sSafetyGate UnlockRequest" := TRUE;
       "ST10_MaterialGate2_DB"."sSafetyGate LockRequest" := FALSE;
       "ST10_SafetyGate_InterfaceDB".H.Status_2 := 2;
   END_IF;
   #_w5 := #_w2 AND ("ST10_SafetyGate_InterfaceDB".H.Status_2 = 3) AND "iMateriel Door Locking FeedBack_H2";
   #_w6 := #_w5 AND NOT "ST10_SafetyGate_InterfaceDB".H.p[3];   // rising edge
   "ST10_SafetyGate_InterfaceDB".H.p[3] := #_w5;
   IF #_w6 THEN
       "ST10_MaterialGate2_DB"."sSafetyGate UnlockRequest" := FALSE;
       "ST10_MaterialGate2_DB"."sSafetyGate LockRequest" := TRUE;
       "ST10_SafetyGate_InterfaceDB".H.Status_2 := 4;
   END_IF;
   IF #_w1 AND ("ST10_SafetyGate_InterfaceDB".H.Status_2 <> 1) AND ("ST10_SafetyGate_InterfaceDB".H.Status_2 <> 2) AND ("ST10_SafetyGate_InterfaceDB".H.Status_2 <> 3) AND ("ST10_SafetyGate_InterfaceDB".H.Status_2 <> 4) THEN
       "ST10_SafetyGate_InterfaceDB".H.Status_2 := 1;
   END_IF;
   IF #_w1 AND ("ST10_SafetyGate_InterfaceDB".H.Status_2 = 2) AND NOT "iShaft_EmptyButton" THEN
       "ST10_SafetyGate_InterfaceDB".H.Status_2 := 3;
   END_IF;
   IF #_w1 AND ("ST10_SafetyGate_InterfaceDB".H.Status_2 = 4) AND NOT "iShaft_EmptyButton" THEN
       "ST10_SafetyGate_InterfaceDB".H.Status_2 := 5;
   END_IF;
END_REGION

REGION Network 18
   RUNG wire#powerrail
      Contact( "AlwaysTRUE" )
      Contact( "AlwaysTRUE" )
      wire#w1
      Contact( "iUnloading_UnlockButton" )
      wire#w2
      { S7_Templates := "SrcType := Int" } EQ_Contact(in1 := "ST10_SafetyGate_InterfaceDB".H.Status_3, in2 := 1)
      P_Trig( "ST10_SafetyGate_InterfaceDB".H.p[10] )
      S_Coil( "ST10_SafetyGate6_DB"."sSafetyGate UnlockRequest" )
      R_Coil( "ST10_SafetyGate6_DB"."sSafetyGate LockRequest" )
      Move(in := 2, out1 => "ST10_SafetyGate_InterfaceDB".H.Status_3)
   END_RUNG
   RUNG wire#w2
      { S7_Templates := "SrcType := Int" } EQ_Contact(in1 := "ST10_SafetyGate_InterfaceDB".H.Status_3, in2 := 3)
      Contact( "iSafety door Locking FeedBack_6" )
      P_Trig( "ST10_SafetyGate_InterfaceDB".H.p[11] )
      R_Coil( "ST10_SafetyGate6_DB"."sSafetyGate UnlockRequest" )
      S_Coil( "ST10_SafetyGate6_DB"."sSafetyGate LockRequest" )
      Move(in := 4, out1 => "ST10_SafetyGate_InterfaceDB".H.Status_3)
   END_RUNG
   RUNG wire#w1
      { S7_Templates := "SrcType := Int" } NE_Contact(in1 := "ST10_SafetyGate_InterfaceDB".H.Status_3, in2 := 1)
      { S7_Templates := "SrcType := Int" } NE_Contact(in1 := "ST10_SafetyGate_InterfaceDB".H.Status_3, in2 := 2)
      { S7_Templates := "SrcType := Int" } NE_Contact(in1 := "ST10_SafetyGate_InterfaceDB".H.Status_3, in2 := 3)
      { S7_Templates := "SrcType := Int" } NE_Contact(in1 := "ST10_SafetyGate_InterfaceDB".H.Status_3, in2 := 4)
      Move(in := 1, out1 => "ST10_SafetyGate_InterfaceDB".H.Status_3)
   END_RUNG
   RUNG wire#w1
      { S7_Templates := "SrcType := Int" } EQ_Contact(in1 := "ST10_SafetyGate_InterfaceDB".H.Status_3, in2 := 2)
      I_Contact( "iUnloading_UnlockButton" )
      Move(in := 3, out1 => "ST10_SafetyGate_InterfaceDB".H.Status_3)
   END_RUNG
   RUNG wire#w1
      { S7_Templates := "SrcType := Int" } EQ_Contact(in1 := "ST10_SafetyGate_InterfaceDB".H.Status_3, in2 := 4)
      I_Contact( "iUnloading_UnlockButton" )
      Move(in := 5, out1 => "ST10_SafetyGate_InterfaceDB".H.Status_3)
   END_RUNG
   // the same network as SCL:
   #_w1 := "AlwaysTRUE" AND "AlwaysTRUE";
   #_w2 := #_w1 AND "iUnloading_UnlockButton";
   #_w3 := #_w2 AND ("ST10_SafetyGate_InterfaceDB".H.Status_3 = 1);
   #_w4 := #_w3 AND NOT "ST10_SafetyGate_InterfaceDB".H.p[10];   // rising edge
   "ST10_SafetyGate_InterfaceDB".H.p[10] := #_w3;
   IF #_w4 THEN
       "ST10_SafetyGate6_DB"."sSafetyGate UnlockRequest" := TRUE;
       "ST10_SafetyGate6_DB"."sSafetyGate LockRequest" := FALSE;
       "ST10_SafetyGate_InterfaceDB".H.Status_3 := 2;
   END_IF;
   #_w5 := #_w2 AND ("ST10_SafetyGate_InterfaceDB".H.Status_3 = 3) AND "iSafety door Locking FeedBack_6";
   #_w6 := #_w5 AND NOT "ST10_SafetyGate_InterfaceDB".H.p[11];   // rising edge
   "ST10_SafetyGate_InterfaceDB".H.p[11] := #_w5;
   IF #_w6 THEN
       "ST10_SafetyGate6_DB"."sSafetyGate UnlockRequest" := FALSE;
       "ST10_SafetyGate6_DB"."sSafetyGate LockRequest" := TRUE;
       "ST10_SafetyGate_InterfaceDB".H.Status_3 := 4;
   END_IF;
   IF #_w1 AND ("ST10_SafetyGate_InterfaceDB".H.Status_3 <> 1) AND ("ST10_SafetyGate_InterfaceDB".H.Status_3 <> 2) AND ("ST10_SafetyGate_InterfaceDB".H.Status_3 <> 3) AND ("ST10_SafetyGate_InterfaceDB".H.Status_3 <> 4) THEN
       "ST10_SafetyGate_InterfaceDB".H.Status_3 := 1;
   END_IF;
   IF #_w1 AND ("ST10_SafetyGate_InterfaceDB".H.Status_3 = 2) AND NOT "iUnloading_UnlockButton" THEN
       "ST10_SafetyGate_InterfaceDB".H.Status_3 := 3;
   END_IF;
   IF #_w1 AND ("ST10_SafetyGate_InterfaceDB".H.Status_3 = 4) AND NOT "iUnloading_UnlockButton" THEN
       "ST10_SafetyGate_InterfaceDB".H.Status_3 := 5;
   END_IF;
END_REGION

REGION Network 19: E-NG料盒-02安全门锁按钮灯
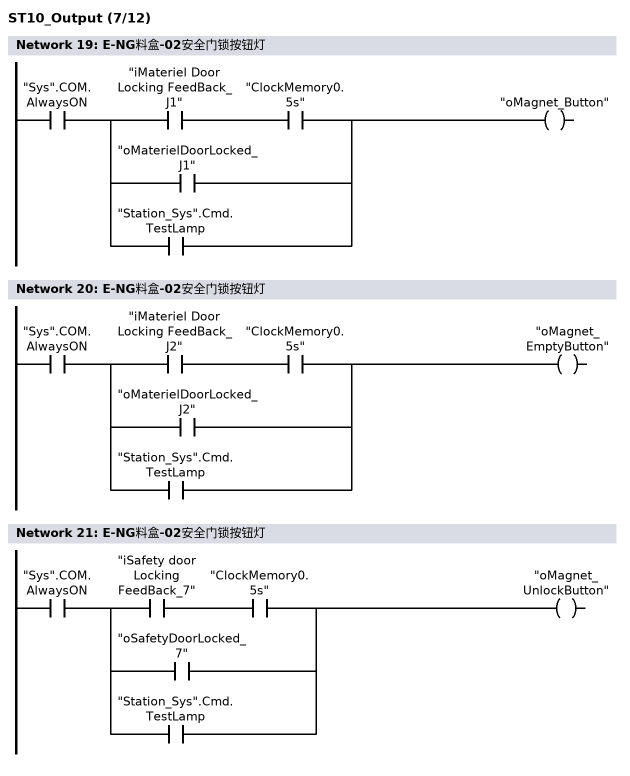
   RUNG wire#powerrail
      Contact( "Sys".COM.AlwaysON )
      wire#w1
      Contact( "iMateriel Door Locking FeedBack_J1" )
      Contact( "ClockMemory0.5s" )
      wire#w2
      Coil( "oMagnet_Button" )
   END_RUNG
   RUNG wire#w1
      Contact( "oMaterielDoorLocked_J1" )
   END_RUNG wire#w2
   RUNG wire#w1
      Contact( "Station_Sys".Cmd.TestLamp )
   END_RUNG wire#w2
   // the same network as SCL:
   "oMagnet_Button" := "Sys".COM.AlwaysON AND (("iMateriel Door Locking FeedBack_J1" AND "ClockMemory0.5s") OR "oMaterielDoorLocked_J1" OR "Station_Sys".Cmd.TestLamp);
END_REGION

REGION Network 20: E-NG料盒-02安全门锁按钮灯
   RUNG wire#powerrail
      Contact( "Sys".COM.AlwaysON )
      wire#w1
      Contact( "iMateriel Door Locking FeedBack_J2" )
      Contact( "ClockMemory0.5s" )
      wire#w2
      Coil( "oMagnet_EmptyButton" )
   END_RUNG
   RUNG wire#w1
      Contact( "oMaterielDoorLocked_J2" )
   END_RUNG wire#w2
   RUNG wire#w1
      Contact( "Station_Sys".Cmd.TestLamp )
   END_RUNG wire#w2
   // the same network as SCL:
   "oMagnet_EmptyButton" := "Sys".COM.AlwaysON AND (("iMateriel Door Locking FeedBack_J2" AND "ClockMemory0.5s") OR "oMaterielDoorLocked_J2" OR "Station_Sys".Cmd.TestLamp);
END_REGION

REGION Network 21: E-NG料盒-02安全门锁按钮灯
   RUNG wire#powerrail
      Contact( "Sys".COM.AlwaysON )
      wire#w1
      Contact( "iSafety door Locking FeedBack_7" )
      Contact( "ClockMemory0.5s" )
      wire#w2
      Coil( "oMagnet_UnlockButton" )
   END_RUNG
   RUNG wire#w1
      Contact( "oSafetyDoorLocked_7" )
   END_RUNG wire#w2
   RUNG wire#w1
      Contact( "Station_Sys".Cmd.TestLamp )
   END_RUNG wire#w2
   // the same network as SCL:
   "oMagnet_UnlockButton" := "Sys".COM.AlwaysON AND (("iSafety door Locking FeedBack_7" AND "ClockMemory0.5s") OR "oSafetyDoorLocked_7" OR "Station_Sys".Cmd.TestLamp);
END_REGION

REGION Network 22
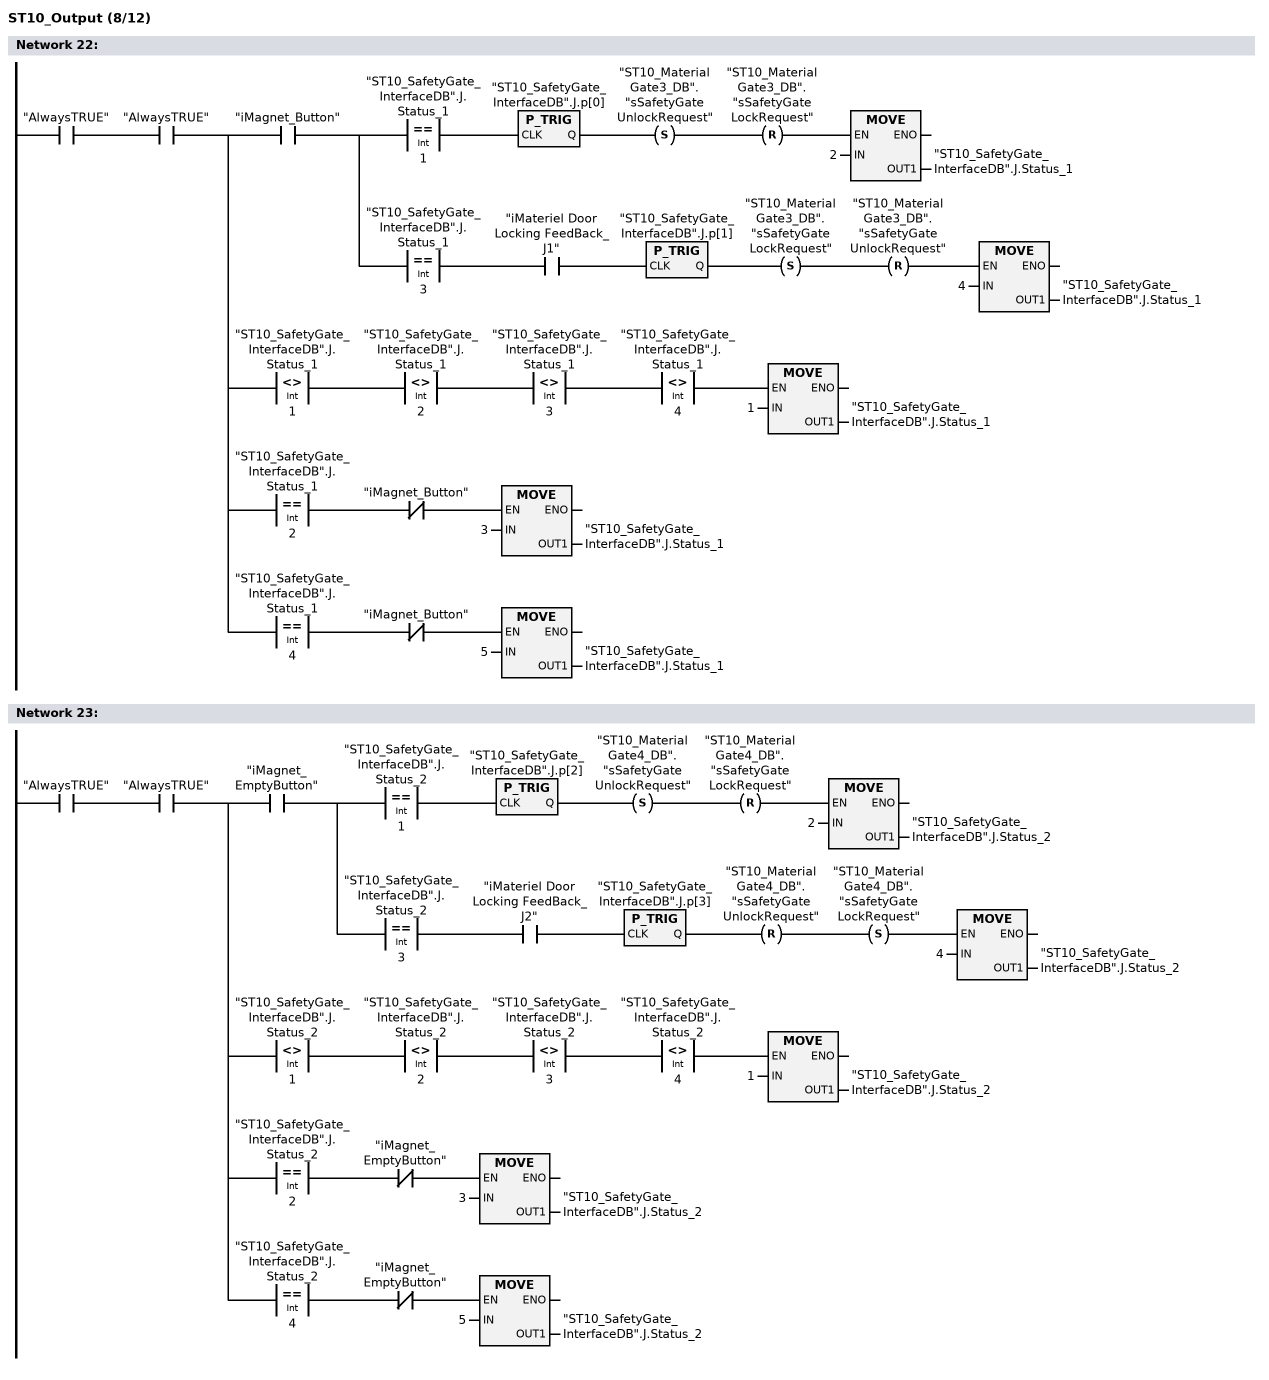
   RUNG wire#powerrail
      Contact( "AlwaysTRUE" )
      Contact( "AlwaysTRUE" )
      wire#w1
      Contact( "iMagnet_Button" )
      wire#w2
      { S7_Templates := "SrcType := Int" } EQ_Contact(in1 := "ST10_SafetyGate_InterfaceDB".J.Status_1, in2 := 1)
      P_Trig( "ST10_SafetyGate_InterfaceDB".J.p[0] )
      S_Coil( "ST10_MaterialGate3_DB"."sSafetyGate UnlockRequest" )
      R_Coil( "ST10_MaterialGate3_DB"."sSafetyGate LockRequest" )
      Move(in := 2, out1 => "ST10_SafetyGate_InterfaceDB".J.Status_1)
   END_RUNG
   RUNG wire#w2
      { S7_Templates := "SrcType := Int" } EQ_Contact(in1 := "ST10_SafetyGate_InterfaceDB".J.Status_1, in2 := 3)
      Contact( "iMateriel Door Locking FeedBack_J1" )
      P_Trig( "ST10_SafetyGate_InterfaceDB".J.p[1] )
      S_Coil( "ST10_MaterialGate3_DB"."sSafetyGate LockRequest" )
      R_Coil( "ST10_MaterialGate3_DB"."sSafetyGate UnlockRequest" )
      Move(in := 4, out1 => "ST10_SafetyGate_InterfaceDB".J.Status_1)
   END_RUNG
   RUNG wire#w1
      { S7_Templates := "SrcType := Int" } NE_Contact(in1 := "ST10_SafetyGate_InterfaceDB".J.Status_1, in2 := 1)
      { S7_Templates := "SrcType := Int" } NE_Contact(in1 := "ST10_SafetyGate_InterfaceDB".J.Status_1, in2 := 2)
      { S7_Templates := "SrcType := Int" } NE_Contact(in1 := "ST10_SafetyGate_InterfaceDB".J.Status_1, in2 := 3)
      { S7_Templates := "SrcType := Int" } NE_Contact(in1 := "ST10_SafetyGate_InterfaceDB".J.Status_1, in2 := 4)
      Move(in := 1, out1 => "ST10_SafetyGate_InterfaceDB".J.Status_1)
   END_RUNG
   RUNG wire#w1
      { S7_Templates := "SrcType := Int" } EQ_Contact(in1 := "ST10_SafetyGate_InterfaceDB".J.Status_1, in2 := 2)
      I_Contact( "iMagnet_Button" )
      Move(in := 3, out1 => "ST10_SafetyGate_InterfaceDB".J.Status_1)
   END_RUNG
   RUNG wire#w1
      { S7_Templates := "SrcType := Int" } EQ_Contact(in1 := "ST10_SafetyGate_InterfaceDB".J.Status_1, in2 := 4)
      I_Contact( "iMagnet_Button" )
      Move(in := 5, out1 => "ST10_SafetyGate_InterfaceDB".J.Status_1)
   END_RUNG
   // the same network as SCL:
   #_w1 := "AlwaysTRUE" AND "AlwaysTRUE";
   #_w2 := #_w1 AND "iMagnet_Button";
   #_w3 := #_w2 AND ("ST10_SafetyGate_InterfaceDB".J.Status_1 = 1);
   #_w4 := #_w3 AND NOT "ST10_SafetyGate_InterfaceDB".J.p[0];   // rising edge
   "ST10_SafetyGate_InterfaceDB".J.p[0] := #_w3;
   IF #_w4 THEN
       "ST10_MaterialGate3_DB"."sSafetyGate UnlockRequest" := TRUE;
       "ST10_MaterialGate3_DB"."sSafetyGate LockRequest" := FALSE;
       "ST10_SafetyGate_InterfaceDB".J.Status_1 := 2;
   END_IF;
   #_w5 := #_w2 AND ("ST10_SafetyGate_InterfaceDB".J.Status_1 = 3) AND "iMateriel Door Locking FeedBack_J1";
   #_w6 := #_w5 AND NOT "ST10_SafetyGate_InterfaceDB".J.p[1];   // rising edge
   "ST10_SafetyGate_InterfaceDB".J.p[1] := #_w5;
   IF #_w6 THEN
       "ST10_MaterialGate3_DB"."sSafetyGate LockRequest" := TRUE;
       "ST10_MaterialGate3_DB"."sSafetyGate UnlockRequest" := FALSE;
       "ST10_SafetyGate_InterfaceDB".J.Status_1 := 4;
   END_IF;
   IF #_w1 AND ("ST10_SafetyGate_InterfaceDB".J.Status_1 <> 1) AND ("ST10_SafetyGate_InterfaceDB".J.Status_1 <> 2) AND ("ST10_SafetyGate_InterfaceDB".J.Status_1 <> 3) AND ("ST10_SafetyGate_InterfaceDB".J.Status_1 <> 4) THEN
       "ST10_SafetyGate_InterfaceDB".J.Status_1 := 1;
   END_IF;
   IF #_w1 AND ("ST10_SafetyGate_InterfaceDB".J.Status_1 = 2) AND NOT "iMagnet_Button" THEN
       "ST10_SafetyGate_InterfaceDB".J.Status_1 := 3;
   END_IF;
   IF #_w1 AND ("ST10_SafetyGate_InterfaceDB".J.Status_1 = 4) AND NOT "iMagnet_Button" THEN
       "ST10_SafetyGate_InterfaceDB".J.Status_1 := 5;
   END_IF;
END_REGION

REGION Network 23
   RUNG wire#powerrail
      Contact( "AlwaysTRUE" )
      Contact( "AlwaysTRUE" )
      wire#w1
      Contact( "iMagnet_EmptyButton" )
      wire#w2
      { S7_Templates := "SrcType := Int" } EQ_Contact(in1 := "ST10_SafetyGate_InterfaceDB".J.Status_2, in2 := 1)
      P_Trig( "ST10_SafetyGate_InterfaceDB".J.p[2] )
      S_Coil( "ST10_MaterialGate4_DB"."sSafetyGate UnlockRequest" )
      R_Coil( "ST10_MaterialGate4_DB"."sSafetyGate LockRequest" )
      Move(in := 2, out1 => "ST10_SafetyGate_InterfaceDB".J.Status_2)
   END_RUNG
   RUNG wire#w2
      { S7_Templates := "SrcType := Int" } EQ_Contact(in1 := "ST10_SafetyGate_InterfaceDB".J.Status_2, in2 := 3)
      Contact( "iMateriel Door Locking FeedBack_J2" )
      P_Trig( "ST10_SafetyGate_InterfaceDB".J.p[3] )
      R_Coil( "ST10_MaterialGate4_DB"."sSafetyGate UnlockRequest" )
      S_Coil( "ST10_MaterialGate4_DB"."sSafetyGate LockRequest" )
      Move(in := 4, out1 => "ST10_SafetyGate_InterfaceDB".J.Status_2)
   END_RUNG
   RUNG wire#w1
      { S7_Templates := "SrcType := Int" } NE_Contact(in1 := "ST10_SafetyGate_InterfaceDB".J.Status_2, in2 := 1)
      { S7_Templates := "SrcType := Int" } NE_Contact(in1 := "ST10_SafetyGate_InterfaceDB".J.Status_2, in2 := 2)
      { S7_Templates := "SrcType := Int" } NE_Contact(in1 := "ST10_SafetyGate_InterfaceDB".J.Status_2, in2 := 3)
      { S7_Templates := "SrcType := Int" } NE_Contact(in1 := "ST10_SafetyGate_InterfaceDB".J.Status_2, in2 := 4)
      Move(in := 1, out1 => "ST10_SafetyGate_InterfaceDB".J.Status_2)
   END_RUNG
   RUNG wire#w1
      { S7_Templates := "SrcType := Int" } EQ_Contact(in1 := "ST10_SafetyGate_InterfaceDB".J.Status_2, in2 := 2)
      I_Contact( "iMagnet_EmptyButton" )
      Move(in := 3, out1 => "ST10_SafetyGate_InterfaceDB".J.Status_2)
   END_RUNG
   RUNG wire#w1
      { S7_Templates := "SrcType := Int" } EQ_Contact(in1 := "ST10_SafetyGate_InterfaceDB".J.Status_2, in2 := 4)
      I_Contact( "iMagnet_EmptyButton" )
      Move(in := 5, out1 => "ST10_SafetyGate_InterfaceDB".J.Status_2)
   END_RUNG
   // the same network as SCL:
   #_w1 := "AlwaysTRUE" AND "AlwaysTRUE";
   #_w2 := #_w1 AND "iMagnet_EmptyButton";
   #_w3 := #_w2 AND ("ST10_SafetyGate_InterfaceDB".J.Status_2 = 1);
   #_w4 := #_w3 AND NOT "ST10_SafetyGate_InterfaceDB".J.p[2];   // rising edge
   "ST10_SafetyGate_InterfaceDB".J.p[2] := #_w3;
   IF #_w4 THEN
       "ST10_MaterialGate4_DB"."sSafetyGate UnlockRequest" := TRUE;
       "ST10_MaterialGate4_DB"."sSafetyGate LockRequest" := FALSE;
       "ST10_SafetyGate_InterfaceDB".J.Status_2 := 2;
   END_IF;
   #_w5 := #_w2 AND ("ST10_SafetyGate_InterfaceDB".J.Status_2 = 3) AND "iMateriel Door Locking FeedBack_J2";
   #_w6 := #_w5 AND NOT "ST10_SafetyGate_InterfaceDB".J.p[3];   // rising edge
   "ST10_SafetyGate_InterfaceDB".J.p[3] := #_w5;
   IF #_w6 THEN
       "ST10_MaterialGate4_DB"."sSafetyGate UnlockRequest" := FALSE;
       "ST10_MaterialGate4_DB"."sSafetyGate LockRequest" := TRUE;
       "ST10_SafetyGate_InterfaceDB".J.Status_2 := 4;
   END_IF;
   IF #_w1 AND ("ST10_SafetyGate_InterfaceDB".J.Status_2 <> 1) AND ("ST10_SafetyGate_InterfaceDB".J.Status_2 <> 2) AND ("ST10_SafetyGate_InterfaceDB".J.Status_2 <> 3) AND ("ST10_SafetyGate_InterfaceDB".J.Status_2 <> 4) THEN
       "ST10_SafetyGate_InterfaceDB".J.Status_2 := 1;
   END_IF;
   IF #_w1 AND ("ST10_SafetyGate_InterfaceDB".J.Status_2 = 2) AND NOT "iMagnet_EmptyButton" THEN
       "ST10_SafetyGate_InterfaceDB".J.Status_2 := 3;
   END_IF;
   IF #_w1 AND ("ST10_SafetyGate_InterfaceDB".J.Status_2 = 4) AND NOT "iMagnet_EmptyButton" THEN
       "ST10_SafetyGate_InterfaceDB".J.Status_2 := 5;
   END_IF;
END_REGION

REGION Network 24
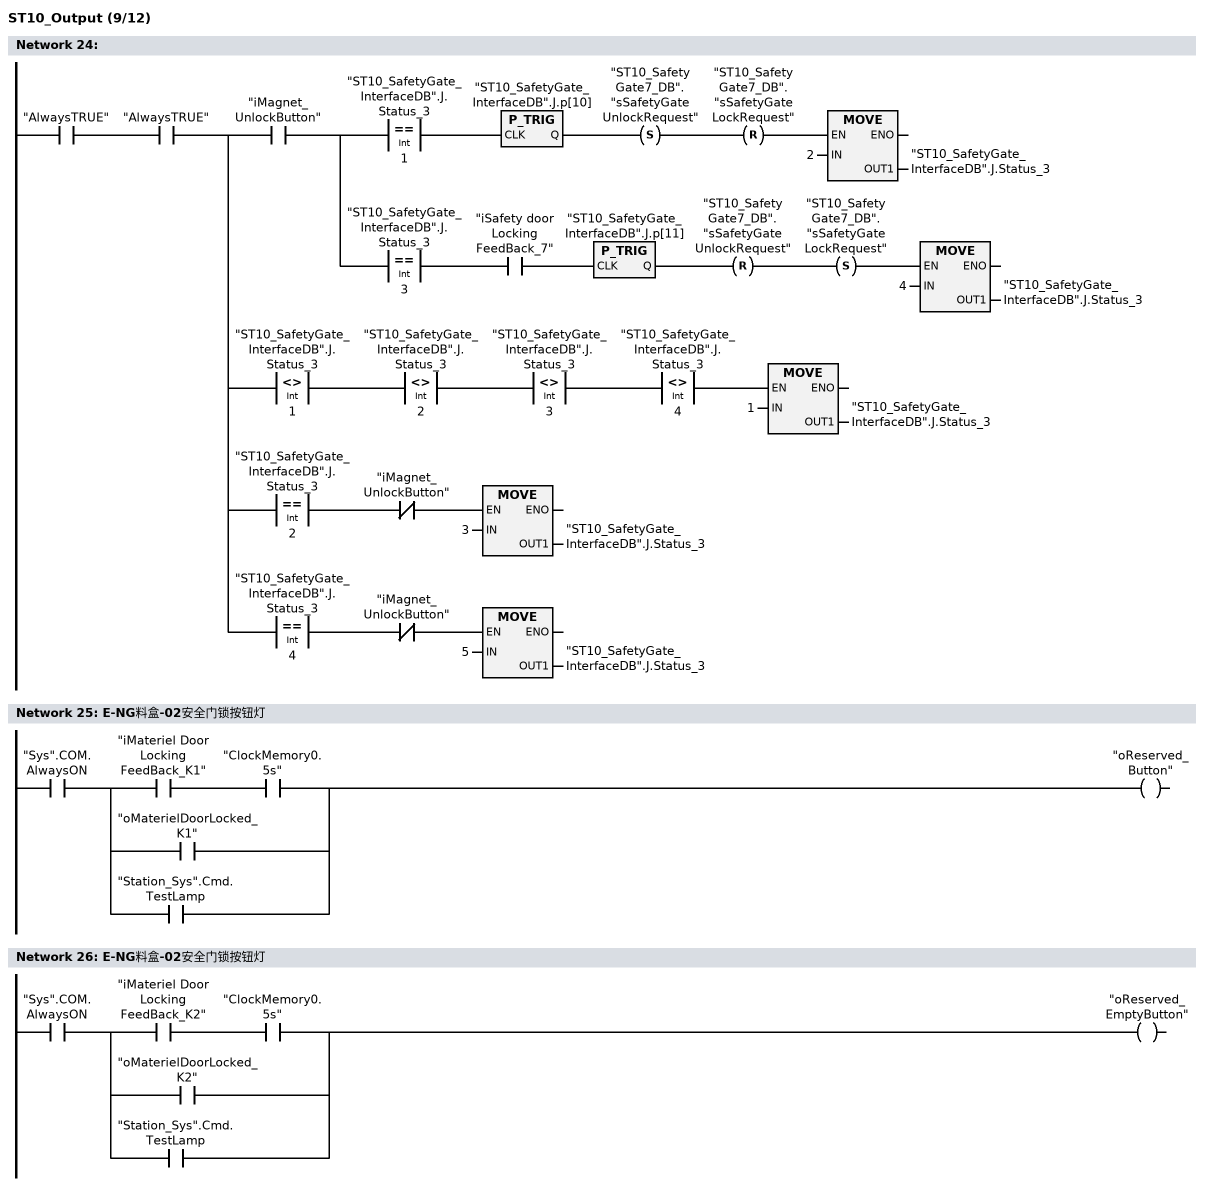
   RUNG wire#powerrail
      Contact( "AlwaysTRUE" )
      Contact( "AlwaysTRUE" )
      wire#w1
      Contact( "iMagnet_UnlockButton" )
      wire#w2
      { S7_Templates := "SrcType := Int" } EQ_Contact(in1 := "ST10_SafetyGate_InterfaceDB".J.Status_3, in2 := 1)
      P_Trig( "ST10_SafetyGate_InterfaceDB".J.p[10] )
      S_Coil( "ST10_SafetyGate7_DB"."sSafetyGate UnlockRequest" )
      R_Coil( "ST10_SafetyGate7_DB"."sSafetyGate LockRequest" )
      Move(in := 2, out1 => "ST10_SafetyGate_InterfaceDB".J.Status_3)
   END_RUNG
   RUNG wire#w2
      { S7_Templates := "SrcType := Int" } EQ_Contact(in1 := "ST10_SafetyGate_InterfaceDB".J.Status_3, in2 := 3)
      Contact( "iSafety door Locking FeedBack_7" )
      P_Trig( "ST10_SafetyGate_InterfaceDB".J.p[11] )
      R_Coil( "ST10_SafetyGate7_DB"."sSafetyGate UnlockRequest" )
      S_Coil( "ST10_SafetyGate7_DB"."sSafetyGate LockRequest" )
      Move(in := 4, out1 => "ST10_SafetyGate_InterfaceDB".J.Status_3)
   END_RUNG
   RUNG wire#w1
      { S7_Templates := "SrcType := Int" } NE_Contact(in1 := "ST10_SafetyGate_InterfaceDB".J.Status_3, in2 := 1)
      { S7_Templates := "SrcType := Int" } NE_Contact(in1 := "ST10_SafetyGate_InterfaceDB".J.Status_3, in2 := 2)
      { S7_Templates := "SrcType := Int" } NE_Contact(in1 := "ST10_SafetyGate_InterfaceDB".J.Status_3, in2 := 3)
      { S7_Templates := "SrcType := Int" } NE_Contact(in1 := "ST10_SafetyGate_InterfaceDB".J.Status_3, in2 := 4)
      Move(in := 1, out1 => "ST10_SafetyGate_InterfaceDB".J.Status_3)
   END_RUNG
   RUNG wire#w1
      { S7_Templates := "SrcType := Int" } EQ_Contact(in1 := "ST10_SafetyGate_InterfaceDB".J.Status_3, in2 := 2)
      I_Contact( "iMagnet_UnlockButton" )
      Move(in := 3, out1 => "ST10_SafetyGate_InterfaceDB".J.Status_3)
   END_RUNG
   RUNG wire#w1
      { S7_Templates := "SrcType := Int" } EQ_Contact(in1 := "ST10_SafetyGate_InterfaceDB".J.Status_3, in2 := 4)
      I_Contact( "iMagnet_UnlockButton" )
      Move(in := 5, out1 => "ST10_SafetyGate_InterfaceDB".J.Status_3)
   END_RUNG
   // the same network as SCL:
   #_w1 := "AlwaysTRUE" AND "AlwaysTRUE";
   #_w2 := #_w1 AND "iMagnet_UnlockButton";
   #_w3 := #_w2 AND ("ST10_SafetyGate_InterfaceDB".J.Status_3 = 1);
   #_w4 := #_w3 AND NOT "ST10_SafetyGate_InterfaceDB".J.p[10];   // rising edge
   "ST10_SafetyGate_InterfaceDB".J.p[10] := #_w3;
   IF #_w4 THEN
       "ST10_SafetyGate7_DB"."sSafetyGate UnlockRequest" := TRUE;
       "ST10_SafetyGate7_DB"."sSafetyGate LockRequest" := FALSE;
       "ST10_SafetyGate_InterfaceDB".J.Status_3 := 2;
   END_IF;
   #_w5 := #_w2 AND ("ST10_SafetyGate_InterfaceDB".J.Status_3 = 3) AND "iSafety door Locking FeedBack_7";
   #_w6 := #_w5 AND NOT "ST10_SafetyGate_InterfaceDB".J.p[11];   // rising edge
   "ST10_SafetyGate_InterfaceDB".J.p[11] := #_w5;
   IF #_w6 THEN
       "ST10_SafetyGate7_DB"."sSafetyGate UnlockRequest" := FALSE;
       "ST10_SafetyGate7_DB"."sSafetyGate LockRequest" := TRUE;
       "ST10_SafetyGate_InterfaceDB".J.Status_3 := 4;
   END_IF;
   IF #_w1 AND ("ST10_SafetyGate_InterfaceDB".J.Status_3 <> 1) AND ("ST10_SafetyGate_InterfaceDB".J.Status_3 <> 2) AND ("ST10_SafetyGate_InterfaceDB".J.Status_3 <> 3) AND ("ST10_SafetyGate_InterfaceDB".J.Status_3 <> 4) THEN
       "ST10_SafetyGate_InterfaceDB".J.Status_3 := 1;
   END_IF;
   IF #_w1 AND ("ST10_SafetyGate_InterfaceDB".J.Status_3 = 2) AND NOT "iMagnet_UnlockButton" THEN
       "ST10_SafetyGate_InterfaceDB".J.Status_3 := 3;
   END_IF;
   IF #_w1 AND ("ST10_SafetyGate_InterfaceDB".J.Status_3 = 4) AND NOT "iMagnet_UnlockButton" THEN
       "ST10_SafetyGate_InterfaceDB".J.Status_3 := 5;
   END_IF;
END_REGION

REGION Network 25: E-NG料盒-02安全门锁按钮灯
   RUNG wire#powerrail
      Contact( "Sys".COM.AlwaysON )
      wire#w1
      Contact( "iMateriel Door Locking FeedBack_K1" )
      Contact( "ClockMemory0.5s" )
      wire#w2
      Coil( "oReserved_Button" )
   END_RUNG
   RUNG wire#w1
      Contact( "oMaterielDoorLocked_K1" )
   END_RUNG wire#w2
   RUNG wire#w1
      Contact( "Station_Sys".Cmd.TestLamp )
   END_RUNG wire#w2
   // the same network as SCL:
   "oReserved_Button" := "Sys".COM.AlwaysON AND (("iMateriel Door Locking FeedBack_K1" AND "ClockMemory0.5s") OR "oMaterielDoorLocked_K1" OR "Station_Sys".Cmd.TestLamp);
END_REGION

REGION Network 26: E-NG料盒-02安全门锁按钮灯
   RUNG wire#powerrail
      Contact( "Sys".COM.AlwaysON )
      wire#w1
      Contact( "iMateriel Door Locking FeedBack_K2" )
      Contact( "ClockMemory0.5s" )
      wire#w2
      Coil( "oReserved_EmptyButton" )
   END_RUNG
   RUNG wire#w1
      Contact( "oMaterielDoorLocked_K2" )
   END_RUNG wire#w2
   RUNG wire#w1
      Contact( "Station_Sys".Cmd.TestLamp )
   END_RUNG wire#w2
   // the same network as SCL:
   "oReserved_EmptyButton" := "Sys".COM.AlwaysON AND (("iMateriel Door Locking FeedBack_K2" AND "ClockMemory0.5s") OR "oMaterielDoorLocked_K2" OR "Station_Sys".Cmd.TestLamp);
END_REGION

REGION Network 27: E-NG料盒-02安全门锁按钮灯
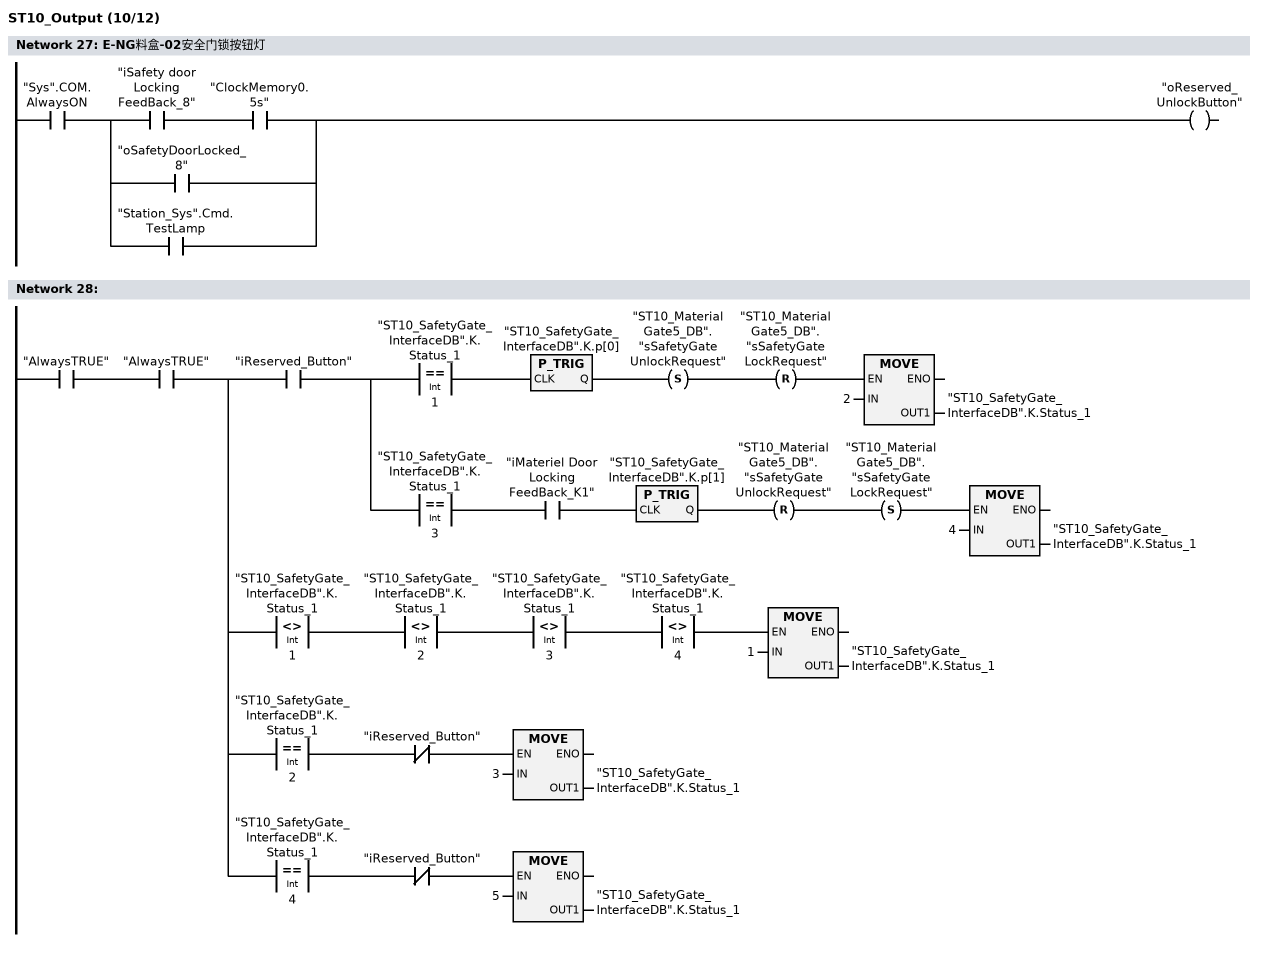
   RUNG wire#powerrail
      Contact( "Sys".COM.AlwaysON )
      wire#w1
      Contact( "iSafety door Locking FeedBack_8" )
      Contact( "ClockMemory0.5s" )
      wire#w2
      Coil( "oReserved_UnlockButton" )
   END_RUNG
   RUNG wire#w1
      Contact( "oSafetyDoorLocked_8" )
   END_RUNG wire#w2
   RUNG wire#w1
      Contact( "Station_Sys".Cmd.TestLamp )
   END_RUNG wire#w2
   // the same network as SCL:
   "oReserved_UnlockButton" := "Sys".COM.AlwaysON AND (("iSafety door Locking FeedBack_8" AND "ClockMemory0.5s") OR "oSafetyDoorLocked_8" OR "Station_Sys".Cmd.TestLamp);
END_REGION

REGION Network 28
   RUNG wire#powerrail
      Contact( "AlwaysTRUE" )
      Contact( "AlwaysTRUE" )
      wire#w1
      Contact( "iReserved_Button" )
      wire#w2
      { S7_Templates := "SrcType := Int" } EQ_Contact(in1 := "ST10_SafetyGate_InterfaceDB".K.Status_1, in2 := 1)
      P_Trig( "ST10_SafetyGate_InterfaceDB".K.p[0] )
      S_Coil( "ST10_MaterialGate5_DB"."sSafetyGate UnlockRequest" )
      R_Coil( "ST10_MaterialGate5_DB"."sSafetyGate LockRequest" )
      Move(in := 2, out1 => "ST10_SafetyGate_InterfaceDB".K.Status_1)
   END_RUNG
   RUNG wire#w2
      { S7_Templates := "SrcType := Int" } EQ_Contact(in1 := "ST10_SafetyGate_InterfaceDB".K.Status_1, in2 := 3)
      Contact( "iMateriel Door Locking FeedBack_K1" )
      P_Trig( "ST10_SafetyGate_InterfaceDB".K.p[1] )
      R_Coil( "ST10_MaterialGate5_DB"."sSafetyGate UnlockRequest" )
      S_Coil( "ST10_MaterialGate5_DB"."sSafetyGate LockRequest" )
      Move(in := 4, out1 => "ST10_SafetyGate_InterfaceDB".K.Status_1)
   END_RUNG
   RUNG wire#w1
      { S7_Templates := "SrcType := Int" } NE_Contact(in1 := "ST10_SafetyGate_InterfaceDB".K.Status_1, in2 := 1)
      { S7_Templates := "SrcType := Int" } NE_Contact(in1 := "ST10_SafetyGate_InterfaceDB".K.Status_1, in2 := 2)
      { S7_Templates := "SrcType := Int" } NE_Contact(in1 := "ST10_SafetyGate_InterfaceDB".K.Status_1, in2 := 3)
      { S7_Templates := "SrcType := Int" } NE_Contact(in1 := "ST10_SafetyGate_InterfaceDB".K.Status_1, in2 := 4)
      Move(in := 1, out1 => "ST10_SafetyGate_InterfaceDB".K.Status_1)
   END_RUNG
   RUNG wire#w1
      { S7_Templates := "SrcType := Int" } EQ_Contact(in1 := "ST10_SafetyGate_InterfaceDB".K.Status_1, in2 := 2)
      I_Contact( "iReserved_Button" )
      Move(in := 3, out1 => "ST10_SafetyGate_InterfaceDB".K.Status_1)
   END_RUNG
   RUNG wire#w1
      { S7_Templates := "SrcType := Int" } EQ_Contact(in1 := "ST10_SafetyGate_InterfaceDB".K.Status_1, in2 := 4)
      I_Contact( "iReserved_Button" )
      Move(in := 5, out1 => "ST10_SafetyGate_InterfaceDB".K.Status_1)
   END_RUNG
   // the same network as SCL:
   #_w1 := "AlwaysTRUE" AND "AlwaysTRUE";
   #_w2 := #_w1 AND "iReserved_Button";
   #_w3 := #_w2 AND ("ST10_SafetyGate_InterfaceDB".K.Status_1 = 1);
   #_w4 := #_w3 AND NOT "ST10_SafetyGate_InterfaceDB".K.p[0];   // rising edge
   "ST10_SafetyGate_InterfaceDB".K.p[0] := #_w3;
   IF #_w4 THEN
       "ST10_MaterialGate5_DB"."sSafetyGate UnlockRequest" := TRUE;
       "ST10_MaterialGate5_DB"."sSafetyGate LockRequest" := FALSE;
       "ST10_SafetyGate_InterfaceDB".K.Status_1 := 2;
   END_IF;
   #_w5 := #_w2 AND ("ST10_SafetyGate_InterfaceDB".K.Status_1 = 3) AND "iMateriel Door Locking FeedBack_K1";
   #_w6 := #_w5 AND NOT "ST10_SafetyGate_InterfaceDB".K.p[1];   // rising edge
   "ST10_SafetyGate_InterfaceDB".K.p[1] := #_w5;
   IF #_w6 THEN
       "ST10_MaterialGate5_DB"."sSafetyGate UnlockRequest" := FALSE;
       "ST10_MaterialGate5_DB"."sSafetyGate LockRequest" := TRUE;
       "ST10_SafetyGate_InterfaceDB".K.Status_1 := 4;
   END_IF;
   IF #_w1 AND ("ST10_SafetyGate_InterfaceDB".K.Status_1 <> 1) AND ("ST10_SafetyGate_InterfaceDB".K.Status_1 <> 2) AND ("ST10_SafetyGate_InterfaceDB".K.Status_1 <> 3) AND ("ST10_SafetyGate_InterfaceDB".K.Status_1 <> 4) THEN
       "ST10_SafetyGate_InterfaceDB".K.Status_1 := 1;
   END_IF;
   IF #_w1 AND ("ST10_SafetyGate_InterfaceDB".K.Status_1 = 2) AND NOT "iReserved_Button" THEN
       "ST10_SafetyGate_InterfaceDB".K.Status_1 := 3;
   END_IF;
   IF #_w1 AND ("ST10_SafetyGate_InterfaceDB".K.Status_1 = 4) AND NOT "iReserved_Button" THEN
       "ST10_SafetyGate_InterfaceDB".K.Status_1 := 5;
   END_IF;
END_REGION

REGION Network 29
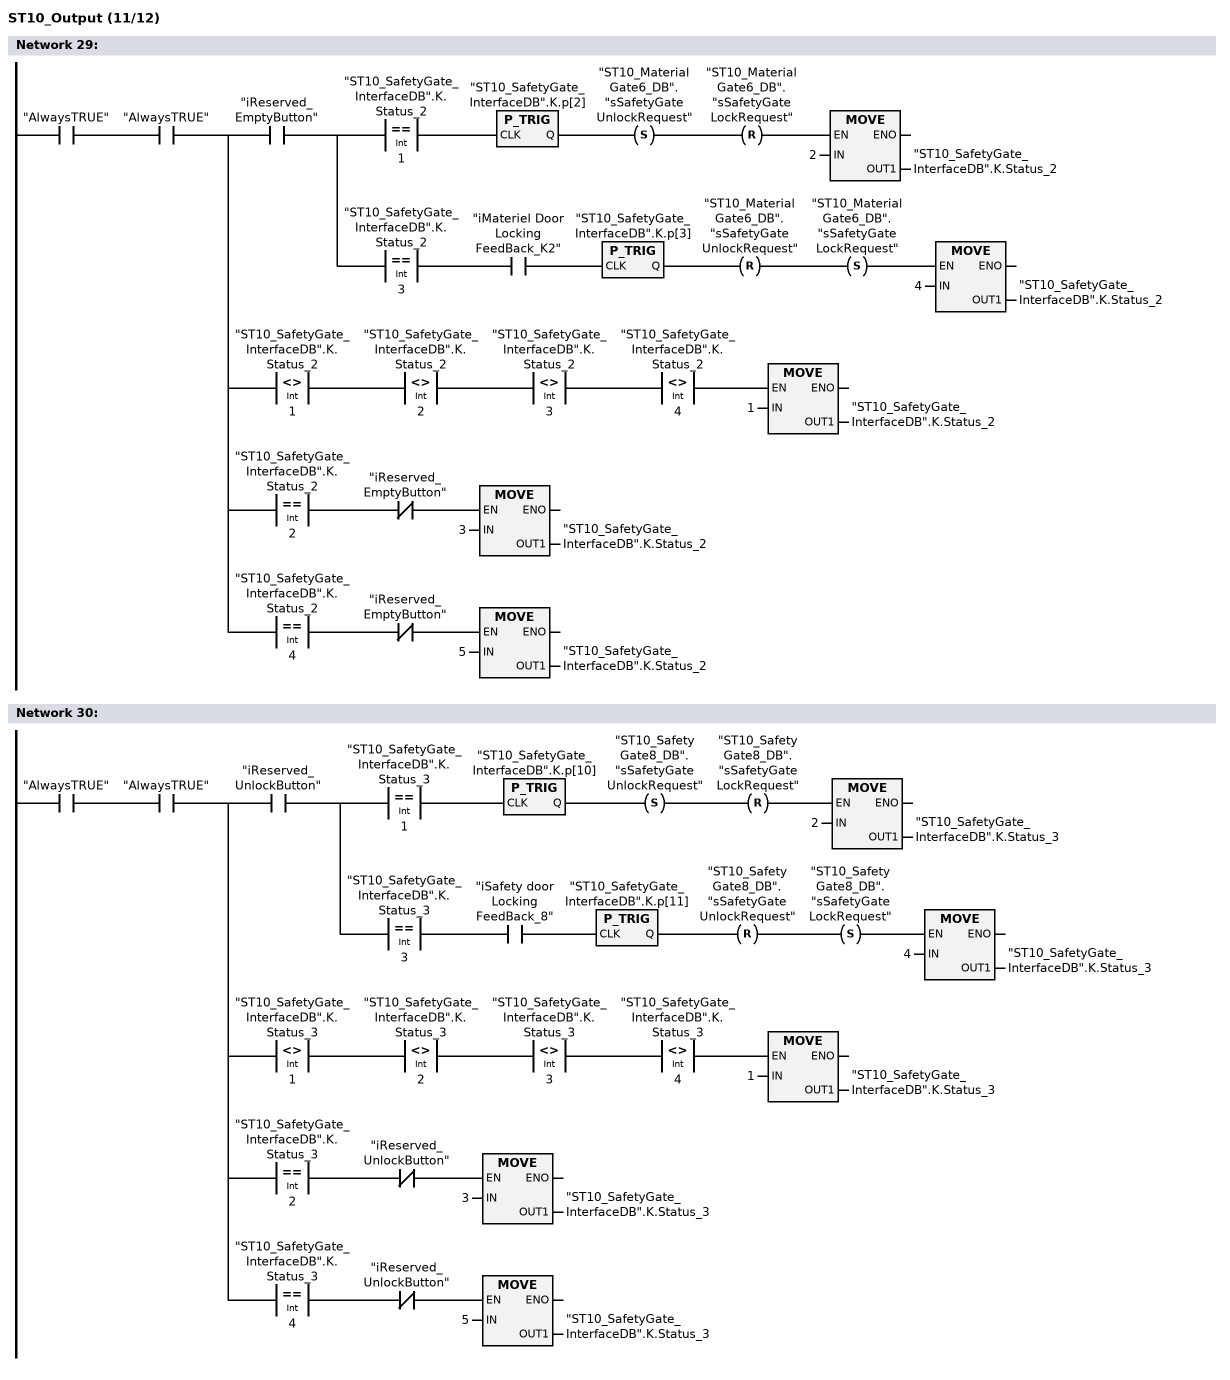
   RUNG wire#powerrail
      Contact( "AlwaysTRUE" )
      Contact( "AlwaysTRUE" )
      wire#w1
      Contact( "iReserved_EmptyButton" )
      wire#w2
      { S7_Templates := "SrcType := Int" } EQ_Contact(in1 := "ST10_SafetyGate_InterfaceDB".K.Status_2, in2 := 1)
      P_Trig( "ST10_SafetyGate_InterfaceDB".K.p[2] )
      S_Coil( "ST10_MaterialGate6_DB"."sSafetyGate UnlockRequest" )
      R_Coil( "ST10_MaterialGate6_DB"."sSafetyGate LockRequest" )
      Move(in := 2, out1 => "ST10_SafetyGate_InterfaceDB".K.Status_2)
   END_RUNG
   RUNG wire#w2
      { S7_Templates := "SrcType := Int" } EQ_Contact(in1 := "ST10_SafetyGate_InterfaceDB".K.Status_2, in2 := 3)
      Contact( "iMateriel Door Locking FeedBack_K2" )
      P_Trig( "ST10_SafetyGate_InterfaceDB".K.p[3] )
      R_Coil( "ST10_MaterialGate6_DB"."sSafetyGate UnlockRequest" )
      S_Coil( "ST10_MaterialGate6_DB"."sSafetyGate LockRequest" )
      Move(in := 4, out1 => "ST10_SafetyGate_InterfaceDB".K.Status_2)
   END_RUNG
   RUNG wire#w1
      { S7_Templates := "SrcType := Int" } NE_Contact(in1 := "ST10_SafetyGate_InterfaceDB".K.Status_2, in2 := 1)
      { S7_Templates := "SrcType := Int" } NE_Contact(in1 := "ST10_SafetyGate_InterfaceDB".K.Status_2, in2 := 2)
      { S7_Templates := "SrcType := Int" } NE_Contact(in1 := "ST10_SafetyGate_InterfaceDB".K.Status_2, in2 := 3)
      { S7_Templates := "SrcType := Int" } NE_Contact(in1 := "ST10_SafetyGate_InterfaceDB".K.Status_2, in2 := 4)
      Move(in := 1, out1 => "ST10_SafetyGate_InterfaceDB".K.Status_2)
   END_RUNG
   RUNG wire#w1
      { S7_Templates := "SrcType := Int" } EQ_Contact(in1 := "ST10_SafetyGate_InterfaceDB".K.Status_2, in2 := 2)
      I_Contact( "iReserved_EmptyButton" )
      Move(in := 3, out1 => "ST10_SafetyGate_InterfaceDB".K.Status_2)
   END_RUNG
   RUNG wire#w1
      { S7_Templates := "SrcType := Int" } EQ_Contact(in1 := "ST10_SafetyGate_InterfaceDB".K.Status_2, in2 := 4)
      I_Contact( "iReserved_EmptyButton" )
      Move(in := 5, out1 => "ST10_SafetyGate_InterfaceDB".K.Status_2)
   END_RUNG
   // the same network as SCL:
   #_w1 := "AlwaysTRUE" AND "AlwaysTRUE";
   #_w2 := #_w1 AND "iReserved_EmptyButton";
   #_w3 := #_w2 AND ("ST10_SafetyGate_InterfaceDB".K.Status_2 = 1);
   #_w4 := #_w3 AND NOT "ST10_SafetyGate_InterfaceDB".K.p[2];   // rising edge
   "ST10_SafetyGate_InterfaceDB".K.p[2] := #_w3;
   IF #_w4 THEN
       "ST10_MaterialGate6_DB"."sSafetyGate UnlockRequest" := TRUE;
       "ST10_MaterialGate6_DB"."sSafetyGate LockRequest" := FALSE;
       "ST10_SafetyGate_InterfaceDB".K.Status_2 := 2;
   END_IF;
   #_w5 := #_w2 AND ("ST10_SafetyGate_InterfaceDB".K.Status_2 = 3) AND "iMateriel Door Locking FeedBack_K2";
   #_w6 := #_w5 AND NOT "ST10_SafetyGate_InterfaceDB".K.p[3];   // rising edge
   "ST10_SafetyGate_InterfaceDB".K.p[3] := #_w5;
   IF #_w6 THEN
       "ST10_MaterialGate6_DB"."sSafetyGate UnlockRequest" := FALSE;
       "ST10_MaterialGate6_DB"."sSafetyGate LockRequest" := TRUE;
       "ST10_SafetyGate_InterfaceDB".K.Status_2 := 4;
   END_IF;
   IF #_w1 AND ("ST10_SafetyGate_InterfaceDB".K.Status_2 <> 1) AND ("ST10_SafetyGate_InterfaceDB".K.Status_2 <> 2) AND ("ST10_SafetyGate_InterfaceDB".K.Status_2 <> 3) AND ("ST10_SafetyGate_InterfaceDB".K.Status_2 <> 4) THEN
       "ST10_SafetyGate_InterfaceDB".K.Status_2 := 1;
   END_IF;
   IF #_w1 AND ("ST10_SafetyGate_InterfaceDB".K.Status_2 = 2) AND NOT "iReserved_EmptyButton" THEN
       "ST10_SafetyGate_InterfaceDB".K.Status_2 := 3;
   END_IF;
   IF #_w1 AND ("ST10_SafetyGate_InterfaceDB".K.Status_2 = 4) AND NOT "iReserved_EmptyButton" THEN
       "ST10_SafetyGate_InterfaceDB".K.Status_2 := 5;
   END_IF;
END_REGION

REGION Network 30
   RUNG wire#powerrail
      Contact( "AlwaysTRUE" )
      Contact( "AlwaysTRUE" )
      wire#w1
      Contact( "iReserved_UnlockButton" )
      wire#w2
      { S7_Templates := "SrcType := Int" } EQ_Contact(in1 := "ST10_SafetyGate_InterfaceDB".K.Status_3, in2 := 1)
      P_Trig( "ST10_SafetyGate_InterfaceDB".K.p[10] )
      S_Coil( "ST10_SafetyGate8_DB"."sSafetyGate UnlockRequest" )
      R_Coil( "ST10_SafetyGate8_DB"."sSafetyGate LockRequest" )
      Move(in := 2, out1 => "ST10_SafetyGate_InterfaceDB".K.Status_3)
   END_RUNG
   RUNG wire#w2
      { S7_Templates := "SrcType := Int" } EQ_Contact(in1 := "ST10_SafetyGate_InterfaceDB".K.Status_3, in2 := 3)
      Contact( "iSafety door Locking FeedBack_8" )
      P_Trig( "ST10_SafetyGate_InterfaceDB".K.p[11] )
      R_Coil( "ST10_SafetyGate8_DB"."sSafetyGate UnlockRequest" )
      S_Coil( "ST10_SafetyGate8_DB"."sSafetyGate LockRequest" )
      Move(in := 4, out1 => "ST10_SafetyGate_InterfaceDB".K.Status_3)
   END_RUNG
   RUNG wire#w1
      { S7_Templates := "SrcType := Int" } NE_Contact(in1 := "ST10_SafetyGate_InterfaceDB".K.Status_3, in2 := 1)
      { S7_Templates := "SrcType := Int" } NE_Contact(in1 := "ST10_SafetyGate_InterfaceDB".K.Status_3, in2 := 2)
      { S7_Templates := "SrcType := Int" } NE_Contact(in1 := "ST10_SafetyGate_InterfaceDB".K.Status_3, in2 := 3)
      { S7_Templates := "SrcType := Int" } NE_Contact(in1 := "ST10_SafetyGate_InterfaceDB".K.Status_3, in2 := 4)
      Move(in := 1, out1 => "ST10_SafetyGate_InterfaceDB".K.Status_3)
   END_RUNG
   RUNG wire#w1
      { S7_Templates := "SrcType := Int" } EQ_Contact(in1 := "ST10_SafetyGate_InterfaceDB".K.Status_3, in2 := 2)
      I_Contact( "iReserved_UnlockButton" )
      Move(in := 3, out1 => "ST10_SafetyGate_InterfaceDB".K.Status_3)
   END_RUNG
   RUNG wire#w1
      { S7_Templates := "SrcType := Int" } EQ_Contact(in1 := "ST10_SafetyGate_InterfaceDB".K.Status_3, in2 := 4)
      I_Contact( "iReserved_UnlockButton" )
      Move(in := 5, out1 => "ST10_SafetyGate_InterfaceDB".K.Status_3)
   END_RUNG
   // the same network as SCL:
   #_w1 := "AlwaysTRUE" AND "AlwaysTRUE";
   #_w2 := #_w1 AND "iReserved_UnlockButton";
   #_w3 := #_w2 AND ("ST10_SafetyGate_InterfaceDB".K.Status_3 = 1);
   #_w4 := #_w3 AND NOT "ST10_SafetyGate_InterfaceDB".K.p[10];   // rising edge
   "ST10_SafetyGate_InterfaceDB".K.p[10] := #_w3;
   IF #_w4 THEN
       "ST10_SafetyGate8_DB"."sSafetyGate UnlockRequest" := TRUE;
       "ST10_SafetyGate8_DB"."sSafetyGate LockRequest" := FALSE;
       "ST10_SafetyGate_InterfaceDB".K.Status_3 := 2;
   END_IF;
   #_w5 := #_w2 AND ("ST10_SafetyGate_InterfaceDB".K.Status_3 = 3) AND "iSafety door Locking FeedBack_8";
   #_w6 := #_w5 AND NOT "ST10_SafetyGate_InterfaceDB".K.p[11];   // rising edge
   "ST10_SafetyGate_InterfaceDB".K.p[11] := #_w5;
   IF #_w6 THEN
       "ST10_SafetyGate8_DB"."sSafetyGate UnlockRequest" := FALSE;
       "ST10_SafetyGate8_DB"."sSafetyGate LockRequest" := TRUE;
       "ST10_SafetyGate_InterfaceDB".K.Status_3 := 4;
   END_IF;
   IF #_w1 AND ("ST10_SafetyGate_InterfaceDB".K.Status_3 <> 1) AND ("ST10_SafetyGate_InterfaceDB".K.Status_3 <> 2) AND ("ST10_SafetyGate_InterfaceDB".K.Status_3 <> 3) AND ("ST10_SafetyGate_InterfaceDB".K.Status_3 <> 4) THEN
       "ST10_SafetyGate_InterfaceDB".K.Status_3 := 1;
   END_IF;
   IF #_w1 AND ("ST10_SafetyGate_InterfaceDB".K.Status_3 = 2) AND NOT "iReserved_UnlockButton" THEN
       "ST10_SafetyGate_InterfaceDB".K.Status_3 := 3;
   END_IF;
   IF #_w1 AND ("ST10_SafetyGate_InterfaceDB".K.Status_3 = 4) AND NOT "iReserved_UnlockButton" THEN
       "ST10_SafetyGate_InterfaceDB".K.Status_3 := 5;
   END_IF;
END_REGION

REGION Network 31: E-NG料盒-02安全门锁按钮灯
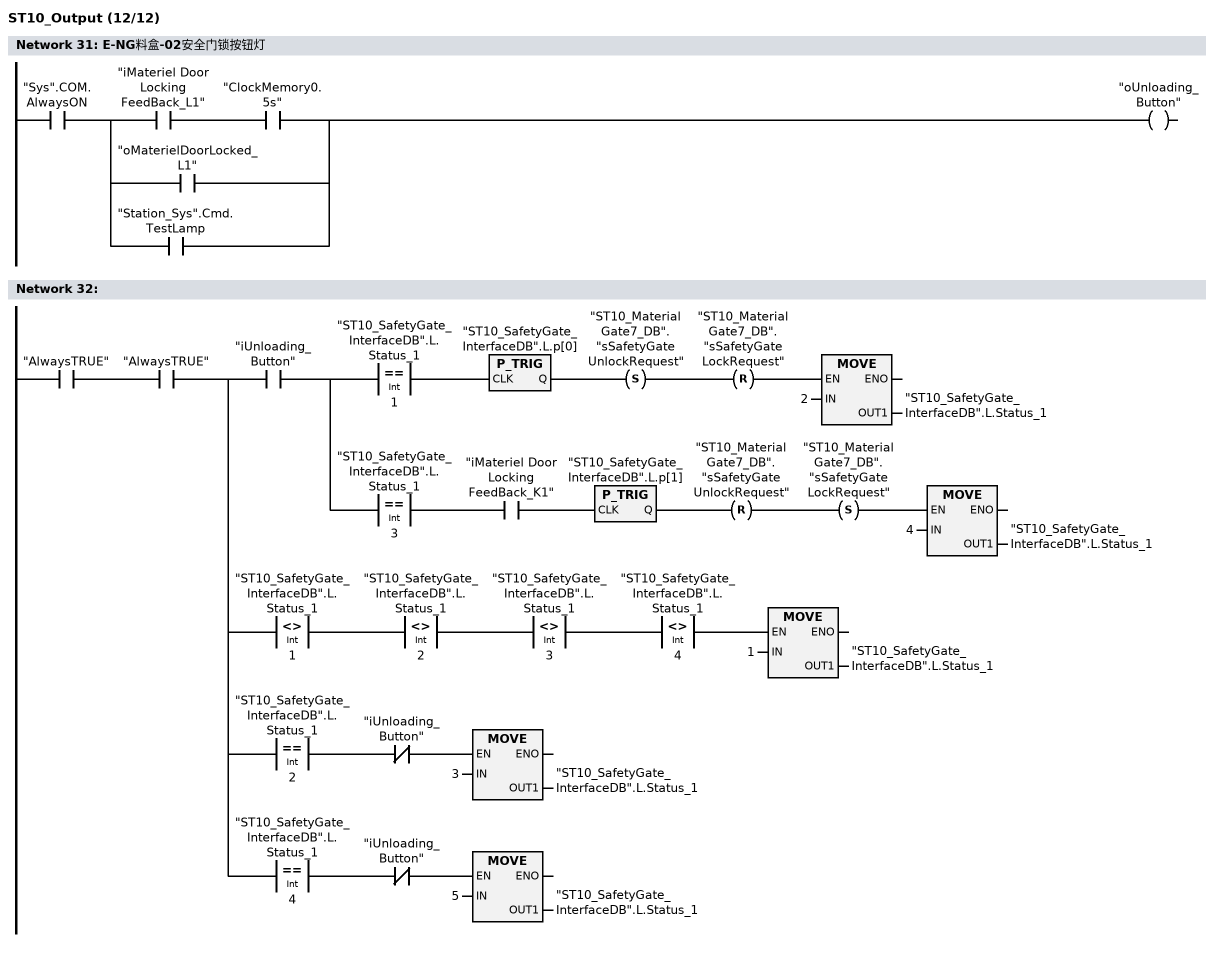
   RUNG wire#powerrail
      Contact( "Sys".COM.AlwaysON )
      wire#w1
      Contact( "iMateriel Door Locking FeedBack_L1" )
      Contact( "ClockMemory0.5s" )
      wire#w2
      Coil( "oUnloading_Button" )
   END_RUNG
   RUNG wire#w1
      Contact( "oMaterielDoorLocked_L1" )
   END_RUNG wire#w2
   RUNG wire#w1
      Contact( "Station_Sys".Cmd.TestLamp )
   END_RUNG wire#w2
   // the same network as SCL:
   "oUnloading_Button" := "Sys".COM.AlwaysON AND (("iMateriel Door Locking FeedBack_L1" AND "ClockMemory0.5s") OR "oMaterielDoorLocked_L1" OR "Station_Sys".Cmd.TestLamp);
END_REGION

REGION Network 32
   RUNG wire#powerrail
      Contact( "AlwaysTRUE" )
      Contact( "AlwaysTRUE" )
      wire#w1
      Contact( "iUnloading_Button" )
      wire#w2
      { S7_Templates := "SrcType := Int" } EQ_Contact(in1 := "ST10_SafetyGate_InterfaceDB".L.Status_1, in2 := 1)
      P_Trig( "ST10_SafetyGate_InterfaceDB".L.p[0] )
      S_Coil( "ST10_MaterialGate7_DB"."sSafetyGate UnlockRequest" )
      R_Coil( "ST10_MaterialGate7_DB"."sSafetyGate LockRequest" )
      Move(in := 2, out1 => "ST10_SafetyGate_InterfaceDB".L.Status_1)
   END_RUNG
   RUNG wire#w2
      { S7_Templates := "SrcType := Int" } EQ_Contact(in1 := "ST10_SafetyGate_InterfaceDB".L.Status_1, in2 := 3)
      Contact( "iMateriel Door Locking FeedBack_K1" )
      P_Trig( "ST10_SafetyGate_InterfaceDB".L.p[1] )
      R_Coil( "ST10_MaterialGate7_DB"."sSafetyGate UnlockRequest" )
      S_Coil( "ST10_MaterialGate7_DB"."sSafetyGate LockRequest" )
      Move(in := 4, out1 => "ST10_SafetyGate_InterfaceDB".L.Status_1)
   END_RUNG
   RUNG wire#w1
      { S7_Templates := "SrcType := Int" } NE_Contact(in1 := "ST10_SafetyGate_InterfaceDB".L.Status_1, in2 := 1)
      { S7_Templates := "SrcType := Int" } NE_Contact(in1 := "ST10_SafetyGate_InterfaceDB".L.Status_1, in2 := 2)
      { S7_Templates := "SrcType := Int" } NE_Contact(in1 := "ST10_SafetyGate_InterfaceDB".L.Status_1, in2 := 3)
      { S7_Templates := "SrcType := Int" } NE_Contact(in1 := "ST10_SafetyGate_InterfaceDB".L.Status_1, in2 := 4)
      Move(in := 1, out1 => "ST10_SafetyGate_InterfaceDB".L.Status_1)
   END_RUNG
   RUNG wire#w1
      { S7_Templates := "SrcType := Int" } EQ_Contact(in1 := "ST10_SafetyGate_InterfaceDB".L.Status_1, in2 := 2)
      I_Contact( "iUnloading_Button" )
      Move(in := 3, out1 => "ST10_SafetyGate_InterfaceDB".L.Status_1)
   END_RUNG
   RUNG wire#w1
      { S7_Templates := "SrcType := Int" } EQ_Contact(in1 := "ST10_SafetyGate_InterfaceDB".L.Status_1, in2 := 4)
      I_Contact( "iUnloading_Button" )
      Move(in := 5, out1 => "ST10_SafetyGate_InterfaceDB".L.Status_1)
   END_RUNG
   // the same network as SCL:
   #_w1 := "AlwaysTRUE" AND "AlwaysTRUE";
   #_w2 := #_w1 AND "iUnloading_Button";
   #_w3 := #_w2 AND ("ST10_SafetyGate_InterfaceDB".L.Status_1 = 1);
   #_w4 := #_w3 AND NOT "ST10_SafetyGate_InterfaceDB".L.p[0];   // rising edge
   "ST10_SafetyGate_InterfaceDB".L.p[0] := #_w3;
   IF #_w4 THEN
       "ST10_MaterialGate7_DB"."sSafetyGate UnlockRequest" := TRUE;
       "ST10_MaterialGate7_DB"."sSafetyGate LockRequest" := FALSE;
       "ST10_SafetyGate_InterfaceDB".L.Status_1 := 2;
   END_IF;
   #_w5 := #_w2 AND ("ST10_SafetyGate_InterfaceDB".L.Status_1 = 3) AND "iMateriel Door Locking FeedBack_K1";
   #_w6 := #_w5 AND NOT "ST10_SafetyGate_InterfaceDB".L.p[1];   // rising edge
   "ST10_SafetyGate_InterfaceDB".L.p[1] := #_w5;
   IF #_w6 THEN
       "ST10_MaterialGate7_DB"."sSafetyGate UnlockRequest" := FALSE;
       "ST10_MaterialGate7_DB"."sSafetyGate LockRequest" := TRUE;
       "ST10_SafetyGate_InterfaceDB".L.Status_1 := 4;
   END_IF;
   IF #_w1 AND ("ST10_SafetyGate_InterfaceDB".L.Status_1 <> 1) AND ("ST10_SafetyGate_InterfaceDB".L.Status_1 <> 2) AND ("ST10_SafetyGate_InterfaceDB".L.Status_1 <> 3) AND ("ST10_SafetyGate_InterfaceDB".L.Status_1 <> 4) THEN
       "ST10_SafetyGate_InterfaceDB".L.Status_1 := 1;
   END_IF;
   IF #_w1 AND ("ST10_SafetyGate_InterfaceDB".L.Status_1 = 2) AND NOT "iUnloading_Button" THEN
       "ST10_SafetyGate_InterfaceDB".L.Status_1 := 3;
   END_IF;
   IF #_w1 AND ("ST10_SafetyGate_InterfaceDB".L.Status_1 = 4) AND NOT "iUnloading_Button" THEN
       "ST10_SafetyGate_InterfaceDB".L.Status_1 := 5;
   END_IF;
END_REGION
END_FUNCTION
